// TwinCAT 3 PLC project Labor_AndreasRies
// ProgramVersion: 3.1.4023.0
// libraries:
//   Lynus Energy Basic, * (Lynus AG)
//   Lynus Persistent Data V1, * (Lynus AG)
//   Lynus Standards, * (Lynus AG)
//   Tc2_IoFunctions, * (Beckhoff Automation GmbH)
//   Tc2_ModbusSrv, * (Beckhoff Automation GmbH)
//   Tc2_Standard, * (Beckhoff Automation GmbH)
//   Tc2_System, * (Beckhoff Automation GmbH)
//   Tc2_Utilities, * (Beckhoff Automation GmbH)
//   Tc3_IotBase, * (Beckhoff Automation GmbH)
//   Tc3_JsonXml, * (Beckhoff Automation GmbH)
//   Tc3_Module, * (Beckhoff Automation GmbH)
//   EfficientIO Communicator,newest,EfficientIO
// project tree:
//   / FastTask.TcTTO, MiddleTask.TcTTO, SlowTask.TcTTO (not stored)
//   FBs/ FB_Shelly_Pro2PM.TcPOU, FB_Shelly_Pro2PM_Helper.TcPOU, FB_Shelly_Pro4PM.TcPOU, FB_Shelly_Pro4PM_Helper.TcPOU
//   POUs/ FB_CurveRead.TcPOU, FB_ECS_Keba_P30.TcPOU, prgComEffIO.TcPOU, prgCS.TcPOU, prgEM.TcPOU, prgMain.TcPOU, prgPersistent.TcPOU, prgRWEffIO.TcPOU, prgVarEffIO.TcPOU, prg_SystemTime.TcPOU
// real-time tasks:
//   TASK FastTask: cycle T#5ms, priority 6, ADS port 350
//   TASK MiddleTask: cycle T#10ms, priority 8, ADS port 351
//   TASK SlowTask: cycle T#20ms, priority 10, ADS port 352
// I/O:
//   DEVICE Gerät 1 (Beckhoff CCAT)
//   DEVICE Gerät 2 (CX-BK)
//     Box 1 (CX-BK)
// variable links:
//   Labor_AndreasRies/Labor_AndreasRies Instance <-> Device 2 (CX-BK)/Box 1 (CX-BK)
//     MiddleTask Inputs/prgEM.fbEM1.fbKL3403.byStateCH1 <-> Term 2 (KL3403)/Channel 1/Status
//     MiddleTask Inputs/prgEM.fbEM1.fbKL3403.byStateCH2 <-> Term 2 (KL3403)/Channel 2/Status
//     MiddleTask Inputs/prgEM.fbEM1.fbKL3403.byStateCH3 <-> Term 2 (KL3403)/Channel 3/Status
//     MiddleTask Inputs/prgEM.fbEM1.fbKL3403.iDataInCH1 <-> Term 2 (KL3403)/Channel 1/Daten Ein
//     MiddleTask Inputs/prgEM.fbEM1.fbKL3403.iDataInCH2 <-> Term 2 (KL3403)/Channel 2/Daten Ein
//     MiddleTask Inputs/prgEM.fbEM1.fbKL3403.iDataInCH3 <-> Term 2 (KL3403)/Channel 3/Daten Ein
//     MiddleTask Inputs/prgEM.fbKBusState.uiKBusState_OUT <-> Inputs/State
//     MiddleTask Inputs/prgMain.int_Temp_1_1 <-> Term 3 (KL3204)/Channel 1/Daten Ein
//     MiddleTask Inputs/prgMain.int_Temp_1_2 <-> Term 3 (KL3204)/Channel 2/Daten Ein
//     MiddleTask Inputs/prgMain.int_Temp_1_3 <-> Term 3 (KL3204)/Channel 3/Daten Ein
//     MiddleTask Inputs/prgMain.int_Temp_1_4 <-> Term 3 (KL3204)/Channel 4/Daten Ein
//     MiddleTask Inputs/prgMain.int_Temp_2_1 <-> Term 4 (KL3204)/Channel 1/Daten Ein
//     MiddleTask Inputs/prgMain.stInData_22/iDataIn <-> Term 4 (KL3204)/Channel 2/Daten Ein
//     MiddleTask Inputs/prgMain.stInData_24/iDataIn <-> Term 4 (KL3204)/Channel 4/Daten Ein
//     MiddleTask Inputs/prgMain.stInData_22/iState <-> Term 4 (KL3204)/Channel 2/Status
//     MiddleTask Inputs/prgMain.stInData_24/iState <-> Term 4 (KL3204)/Channel 4/Status
//     MiddleTask Inputs/prgMain.stInData_W22/iDataIn <-> Term 4 (KL3204)/Channel 3/Daten Ein
//     MiddleTask Inputs/prgMain.stInData_W22/iState <-> Term 4 (KL3204)/Channel 3/Status
//     MiddleTask Outputs/prgEM.fbEM1.fbKL3403.byCntrCH1 <-> Term 2 (KL3403)/Channel 1/Kontrolle
//     MiddleTask Outputs/prgEM.fbEM1.fbKL3403.byCntrCH2 <-> Term 2 (KL3403)/Channel 2/Kontrolle
//     MiddleTask Outputs/prgEM.fbEM1.fbKL3403.byCntrCH3 <-> Term 2 (KL3403)/Channel 3/Kontrolle
//     MiddleTask Outputs/prgMain.stOutData_22/iCtrl <-> Term 4 (KL3204)/Channel 2/Kontrolle
//     MiddleTask Outputs/prgMain.stOutData_24/iCtrl <-> Term 4 (KL3204)/Channel 4/Kontrolle
//     MiddleTask Outputs/prgMain.stOutData_22/iDataOut <-> Term 4 (KL3204)/Channel 2/Daten Aus
//     MiddleTask Outputs/prgMain.stOutData_24/iDataOut <-> Term 4 (KL3204)/Channel 4/Daten Aus
//     MiddleTask Outputs/prgMain.stOutData_W22/iCtrl <-> Term 4 (KL3204)/Channel 3/Kontrolle
//     MiddleTask Outputs/prgMain.stOutData_W22/iDataOut <-> Term 4 (KL3204)/Channel 3/Daten Aus

CONFIGURATION Labor_AndreasRies
    RESOURCE PLC ON TwinCAT3
        TASK FastTask(INTERVAL := T#5ms, PRIORITY := 6);
        TASK MiddleTask(INTERVAL := T#10ms, PRIORITY := 8);
        PROGRAM prgRWEffIO WITH FastTask : prgRWEffIO;
        PROGRAM prgVarEffIO WITH FastTask : prgVarEffIO;
        PROGRAM prg_SystemTime WITH FastTask : prg_SystemTime;
        PROGRAM prgCS WITH MiddleTask : prgCS;
        PROGRAM prgEM WITH MiddleTask : prgEM;
        PROGRAM prgPersistent WITH MiddleTask : prgPersistent;
        PROGRAM prgMain WITH MiddleTask : prgMain;
    END_RESOURCE
END_CONFIGURATION

// ---- POUs/prgRWEffIO.TcPOU
PROGRAM prgRWEffIO
VAR
	fbRW1		: FB_ReadWrite_V2;
	mFirst: BOOL;
END_VAR

fbRW1(bBusy=> , bError=> , udiErrorCodeOut=> , eErrorReadWrite_Out=> );


IF mFirst=FALSE THEN
	prgRWEffIO.fbRW1.eUploadType := 4;
	mFirst:=TRUE;	
END_IF

END_PROGRAM

// ---- POUs/prgVarEffIO.TcPOU
PROGRAM prgVarEffIO
VAR
	fbVar		: FB_VarInfo;
	int_temp_1	:INT; 					//{#lynus.ag#()}
	int_temp_2	:INT; 					//{#lynus.ag#()}
	int_temp_3	:INT; 					//{#lynus.ag#()}
	int_temp_4	:INT; 					//{#lynus.ag#()}
	int_temp_5	:INT; 					//{#lynus.ag#()}
	int_temp_6	:INT; 					//{#lynus.ag#()}
	int_temp_7	:INT; 					//{#lynus.ag#()}
	int_temp_8	:INT; 					//{#lynus.ag#()}
	int_temp_9	:INT; 					//{#lynus.ag#()}
	int_temp_10	:INT; 					//{#lynus.ag#()}
	int_temp_11	:INT; 					//{#lynus.ag#()}
	int_temp_12	:INT; 					//{#lynus.ag#()}
	int_temp_13	:INT; 					//{#lynus.ag#()}
	int_temp_14	:INT; 					//{#lynus.ag#()}
	int_temp_15	:INT; 					//{#lynus.ag#()}
	int_temp_16	:INT; 					//{#lynus.ag#()}
	int_temp_17	:INT; 					//{#lynus.ag#()}
	int_temp_18	:INT; 					//{#lynus.ag#()}
	int_temp_19	:INT; 					//{#lynus.ag#()}
	int_temp_20	:INT; 					//{#lynus.ag#()}
	int_temp_21	:INT; 					//{#lynus.ag#()}
	int_temp_22	:INT; 					//{#lynus.ag#()}
	int_temp_23	:INT; 					//{#lynus.ag#()}
	int_temp_24	:INT; 					//{#lynus.ag#()}
	int_temp_25	:INT; 					//{#lynus.ag#()}
	int_temp_26	:INT; 					//{#lynus.ag#()}
	int_temp_27	:INT; 					//{#lynus.ag#()}
	int_temp_28	:INT; 					//{#lynus.ag#()}
	int_temp_29	:INT; 					//{#lynus.ag#()}
	int_temp_30	:INT; 					//{#lynus.ag#()}
	int_temp_31	:INT; 					//{#lynus.ag#()}
	int_temp_32	:INT; 					//{#lynus.ag#()}
	int_temp_33	:INT; 					//{#lynus.ag#()}
	int_temp_34	:INT; 					//{#lynus.ag#()}
	int_temp_35	:INT; 					//{#lynus.ag#()}
	int_temp_36	:INT; 					//{#lynus.ag#()}
	int_temp_37	:INT; 					//{#lynus.ag#()}
	int_temp_38	:INT; 					//{#lynus.ag#()}
	int_temp_39	:INT; 					//{#lynus.ag#()}
	int_temp_40	:INT; 					//{#lynus.ag#()}
	int_temp_41	:INT; 					//{#lynus.ag#()}
	int_temp_42	:INT; 					//{#lynus.ag#()}
	int_temp_43	:INT; 					//{#lynus.ag#()}
	int_temp_44	:INT; 					//{#lynus.ag#()}
	int_temp_45	:INT; 					//{#lynus.ag#()}
	int_temp_46	:INT; 					//{#lynus.ag#()}
	int_temp_47	:INT; 					//{#lynus.ag#()}
	int_temp_48	:INT; 					//{#lynus.ag#()}
	int_temp_49	:INT; 					//{#lynus.ag#()}
	int_temp2_1	:INT; 					//{#lynus.ag#()}
	int_temp2_2	:INT; 					//{#lynus.ag#()}
	int_temp2_3	:INT; 					//{#lynus.ag#()}
	int_temp2_4	:INT; 					//{#lynus.ag#()}
	int_temp2_5	:INT; 					//{#lynus.ag#()}
	int_temp2_6	:INT; 					//{#lynus.ag#()}
	int_temp2_7	:INT; 					//{#lynus.ag#()}
	int_temp2_8	:INT; 					//{#lynus.ag#()}
	int_temp2_9	:INT; 					//{#lynus.ag#()}
	int_temp2_10	:INT; 					//{#lynus.ag#()}
	int_temp2_11	:INT; 					//{#lynus.ag#()}
	int_temp2_12	:INT; 					//{#lynus.ag#()}
	int_temp2_13	:INT; 					//{#lynus.ag#()}
	int_temp2_14	:INT; 					//{#lynus.ag#()}
	int_temp2_15	:INT; 					//{#lynus.ag#()}
	int_temp2_16	:INT; 					//{#lynus.ag#()}
	int_temp2_17	:INT; 					//{#lynus.ag#()}
	int_temp2_18	:INT; 					//{#lynus.ag#()}
	int_temp2_19	:INT; 					//{#lynus.ag#()}
	int_temp2_20	:INT; 					//{#lynus.ag#()}
	int_temp2_21	:INT; 					//{#lynus.ag#()}
	int_temp2_22	:INT; 					//{#lynus.ag#()}
	int_temp2_23	:INT; 					//{#lynus.ag#()}
	int_temp2_24	:INT; 					//{#lynus.ag#()}
	int_temp2_25	:INT; 					//{#lynus.ag#()}
	int_temp2_26	:INT; 					//{#lynus.ag#()}
	int_temp2_27	:INT; 					//{#lynus.ag#()}
	int_temp2_28	:INT; 					//{#lynus.ag#()}
	int_temp2_29	:INT; 					//{#lynus.ag#()}
	int_temp2_30	:INT; 					//{#lynus.ag#()}
	int_temp2_31	:INT; 					//{#lynus.ag#()}
	int_temp2_32	:INT; 					//{#lynus.ag#()}
	int_temp2_33	:INT; 					//{#lynus.ag#()}
	int_temp2_34	:INT; 					//{#lynus.ag#()}
	int_temp2_35	:INT; 					//{#lynus.ag#()}
	int_temp2_36	:INT; 					//{#lynus.ag#()}
	int_temp2_37	:INT; 					//{#lynus.ag#()}
	int_temp2_38	:INT; 					//{#lynus.ag#()}
	int_temp2_39	:INT; 					//{#lynus.ag#()}
	int_temp2_40	:INT; 					//{#lynus.ag#()}
	int_temp2_41	:INT; 					//{#lynus.ag#()}
	int_temp2_42	:INT; 					//{#lynus.ag#()}
	int_temp2_43	:INT; 					//{#lynus.ag#()}
	int_temp2_44	:INT; 					//{#lynus.ag#()}
	int_temp2_45	:INT; 					//{#lynus.ag#()}
	int_temp2_46	:INT; 					//{#lynus.ag#()}
	int_temp2_47	:INT; 					//{#lynus.ag#()}
	int_temp2_48	:INT; 					//{#lynus.ag#()}
	int_temp2_49	:INT; 					//{#lynus.ag#()}
	int_temp3_1	:INT; 					//{#lynus.ag#()}
	int_temp3_2	:INT; 					//{#lynus.ag#()}
	int_temp3_3	:INT; 					//{#lynus.ag#()}
	int_temp3_4	:INT; 					//{#lynus.ag#()}
	int_temp3_5	:INT; 					//{#lynus.ag#()}
	int_temp3_6	:INT; 					//{#lynus.ag#()}
	int_temp3_7	:INT; 					//{#lynus.ag#()}
	int_temp3_8	:INT; 					//{#lynus.ag#()}
	int_temp3_9	:INT; 					//{#lynus.ag#()}
	int_temp3_10	:INT; 					//{#lynus.ag#()}
	int_temp3_11	:INT; 					//{#lynus.ag#()}
	int_temp3_12	:INT; 					//{#lynus.ag#()}
	int_temp3_13	:INT; 					//{#lynus.ag#()}
	int_temp3_14	:INT; 					//{#lynus.ag#()}
	int_temp3_15	:INT; 					//{#lynus.ag#()}
	int_temp3_16	:INT; 					//{#lynus.ag#()}
	int_temp3_17	:INT; 					//{#lynus.ag#()}
	int_temp3_18	:INT; 					//{#lynus.ag#()}
	int_temp3_19	:INT; 					//{#lynus.ag#()}
	int_temp3_20	:INT; 					//{#lynus.ag#()}
	int_temp3_21	:INT; 					//{#lynus.ag#()}
	int_temp3_22	:INT; 					//{#lynus.ag#()}
	int_temp3_23	:INT; 					//{#lynus.ag#()}
	int_temp3_24	:INT; 					//{#lynus.ag#()}
	int_temp3_25	:INT; 					//{#lynus.ag#()}
	int_temp3_26	:INT; 					//{#lynus.ag#()}
	int_temp3_27	:INT; 					//{#lynus.ag#()}
	int_temp3_28	:INT; 					//{#lynus.ag#()}
	int_temp3_29	:INT; 					//{#lynus.ag#()}
	int_temp3_30	:INT; 					//{#lynus.ag#()}
	int_temp3_31	:INT; 					//{#lynus.ag#()}
	int_temp3_32	:INT; 					//{#lynus.ag#()}
	int_temp3_33	:INT; 					//{#lynus.ag#()}
	int_temp3_34	:INT; 					//{#lynus.ag#()}
	int_temp3_35	:INT; 					//{#lynus.ag#()}
	int_temp3_36	:INT; 					//{#lynus.ag#()}
	int_temp3_37	:INT; 					//{#lynus.ag#()}
	int_temp3_38	:INT; 					//{#lynus.ag#()}
	int_temp3_39	:INT; 					//{#lynus.ag#()}
	int_temp3_40	:INT; 					//{#lynus.ag#()}
	int_temp3_41	:INT; 					//{#lynus.ag#()}
	int_temp3_42	:INT; 					//{#lynus.ag#()}
	int_temp3_43	:INT; 					//{#lynus.ag#()}
	int_temp3_44	:INT; 					//{#lynus.ag#()}
	int_temp3_45	:INT; 					//{#lynus.ag#()}
	int_temp3_46	:INT; 					//{#lynus.ag#()}
	int_temp3_47	:INT; 					//{#lynus.ag#()}
	int_temp3_48	:INT; 					//{#lynus.ag#()}
	int_temp3_49	:INT; 					//{#lynus.ag#()}
	int_temp4_1	:INT; 					//{#lynus.ag#()}
	int_temp4_2	:INT; 					//{#lynus.ag#()}
	int_temp4_3	:INT; 					//{#lynus.ag#()}
	int_temp4_4	:INT; 					//{#lynus.ag#()}
	int_temp4_5	:INT; 					//{#lynus.ag#()}
	int_temp4_6	:INT; 					//{#lynus.ag#()}
	int_temp4_7	:INT; 					//{#lynus.ag#()}
	int_temp4_8	:INT; 					//{#lynus.ag#()}
	int_temp4_9	:INT; 					//{#lynus.ag#()}
	int_temp4_10	:INT; 					//{#lynus.ag#()}
	int_temp4_11	:INT; 					//{#lynus.ag#()}
	int_temp4_12	:INT; 					//{#lynus.ag#()}
	int_temp4_13	:INT; 					//{#lynus.ag#()}
	int_temp4_14	:INT; 					//{#lynus.ag#()}
	int_temp4_15	:INT; 					//{#lynus.ag#()}
	int_temp4_16	:INT; 					//{#lynus.ag#()}
	int_temp4_17	:INT; 					//{#lynus.ag#()}
	int_temp4_18	:INT; 					//{#lynus.ag#()}
	int_temp4_19	:INT; 					//{#lynus.ag#()}
	int_temp4_20	:INT; 					//{#lynus.ag#()}
	int_temp4_21	:INT; 					//{#lynus.ag#()}
	int_temp4_22	:INT; 					//{#lynus.ag#()}
	int_temp4_23	:INT; 					//{#lynus.ag#()}
	int_temp4_24	:INT; 					//{#lynus.ag#()}
	int_temp4_25	:INT; 					//{#lynus.ag#()}
	int_temp4_26	:INT; 					//{#lynus.ag#()}
	int_temp4_27	:INT; 					//{#lynus.ag#()}
	int_temp4_28	:INT; 					//{#lynus.ag#()}
	int_temp4_29	:INT; 					//{#lynus.ag#()}
	int_temp4_30	:INT; 					//{#lynus.ag#()}
	int_temp4_31	:INT; 					//{#lynus.ag#()}
	int_temp4_32	:INT; 					//{#lynus.ag#()}
	int_temp4_33	:INT; 					//{#lynus.ag#()}
	int_temp4_34	:INT; 					//{#lynus.ag#()}
	int_temp4_35	:INT; 					//{#lynus.ag#()}
	int_temp4_36	:INT; 					//{#lynus.ag#()}
	int_temp4_37	:INT; 					//{#lynus.ag#()}
	int_temp4_38	:INT; 					//{#lynus.ag#()}
	int_temp4_39	:INT; 					//{#lynus.ag#()}
	int_temp4_40	:INT; 					//{#lynus.ag#()}
	int_temp4_41	:INT; 					//{#lynus.ag#()}
	int_temp4_42	:INT; 					//{#lynus.ag#()}
	int_temp4_43	:INT; 					//{#lynus.ag#()}
	int_temp4_44	:INT; 					//{#lynus.ag#()}
	int_temp4_45	:INT; 					//{#lynus.ag#()}
	int_temp4_46	:INT; 					//{#lynus.ag#()}
	int_temp4_47	:INT; 					//{#lynus.ag#()}
	int_temp4_48	:INT; 					//{#lynus.ag#()}
	int_temp4_49	:INT; 					//{#lynus.ag#()}
	m_test: BOOL;
	mtest: BOOL;
END_VAR

fbVar(
	bReadInfo:= , 
	eTMCFile:= eSelectTMCFile.eDontUseTMCFile, 
	eSavePositionTMCFile:= eSavePositionOnPLC.ePostionHardDisk, 
	udiCounterFoundVariables=> , 
	bError=> , 
	bBusy=> , 
	byProgress=> , 
	udiErrorCodeOut=> , 
	eErrorVarInfo_Out=> , 
	sVarWithError=> );
IF mtest THEN
	int_temp_1 := 	int_temp_1+1;
	int_temp_2 := 	int_temp_2+10;
	int_temp_3 := 	int_temp_3+100;
	int_temp_4 := 	int_temp_4+1000;
	int_temp_5 := 	int_temp_5-1;
	int_temp_6 := 	int_temp_6-10;
	int_temp_7 := 	int_temp_7-100;
	int_temp_8 := 	int_temp_8-1000;
	int_temp_9 := 	int_temp_9+2;
	int_temp_10 := 	int_temp_10+5;
	int_temp_11 := 	int_temp_1;
	int_temp_12 := 	int_temp_2;
	int_temp_13 := 	int_temp_3;
	int_temp_14 := 	int_temp_4;
	int_temp_15 := 	int_temp_5;
	int_temp_16 := 	int_temp_6;
	int_temp_17 := 	int_temp_7;
	int_temp_18 := 	int_temp_8;
	int_temp_19 := 	int_temp_9;
	int_temp_20 := 	int_temp_10;
	int_temp_21 := 	int_temp_1;
	int_temp_22 := 	int_temp_2;
	int_temp_23 := 	int_temp_3;
	int_temp_24 := 	int_temp_4;
	int_temp_25 := 	int_temp_5;
	int_temp_26 := 	int_temp_6;
	int_temp_27 := 	int_temp_7;
	int_temp_28 := 	int_temp_8;
	int_temp_29 := 	int_temp_9;
	int_temp_30 := 	int_temp_10;
	int_temp_31 := 	int_temp_1;
	int_temp_32 := 	int_temp_2;
	int_temp_33 := 	int_temp_3;
	int_temp_34 := 	int_temp_4;
	int_temp_35 := 	int_temp_5;
	int_temp_36 := 	int_temp_6;
	int_temp_37 := 	int_temp_7;
	int_temp_38 := 	int_temp_8;
	int_temp_39 := 	int_temp_9;
	int_temp_40 := 	int_temp_10;
	int_temp_41 := 	int_temp_1;
	int_temp_42 := 	int_temp_2;
	int_temp_43 := 	int_temp_3;
	int_temp_44 := 	int_temp_4;
	int_temp_45 := 	int_temp_5;
	int_temp_46 := 	int_temp_6;
	int_temp_47 := 	int_temp_7;
	int_temp_48 := 	int_temp_8;
	int_temp_49 := 	int_temp_9;
	int_temp2_1 := 	int_temp2_1+1;
	int_temp2_2 := 	int_temp2_2+10;
	int_temp2_3 := 	int_temp2_3+100;
	int_temp2_4 := 	int_temp2_4+1000;
	int_temp2_5 := 	int_temp2_5-1;
	int_temp2_6 := 	int_temp2_6-10;
	int_temp2_7 := 	int_temp2_7-100;
	int_temp2_8 := 	int_temp2_8-1000;
	int_temp2_9 := 	int_temp2_9+2;
	int_temp2_10 := 	int_temp2_10+5;
	int_temp2_11 := 	int_temp2_1;
	int_temp2_12 := 	int_temp2_2;
	int_temp2_13 := 	int_temp2_3;
	int_temp2_14 := 	int_temp2_4;
	int_temp2_15 := 	int_temp2_5;
	int_temp2_16 := 	int_temp2_6;
	int_temp2_17 := 	int_temp2_7;
	int_temp2_18 := 	int_temp2_8;
	int_temp2_19 := 	int_temp2_9;
	int_temp2_20 := 	int_temp2_10;
	int_temp2_21 := 	int_temp2_1;
	int_temp2_22 := 	int_temp2_2;
	int_temp2_23 := 	int_temp2_3;
	int_temp2_24 := 	int_temp2_4;
	int_temp2_25 := 	int_temp2_5;
	int_temp2_26 := 	int_temp2_6;
	int_temp2_27 := 	int_temp2_7;
	int_temp2_28 := 	int_temp2_8;
	int_temp2_29 := 	int_temp2_9;
	int_temp2_30 := 	int_temp2_10;
	int_temp2_31 := 	int_temp2_1;
	int_temp2_32 := 	int_temp2_2;
	int_temp2_33 := 	int_temp2_3;
	int_temp2_34 := 	int_temp2_4;
	int_temp2_35 := 	int_temp2_5;
	int_temp2_36 := 	int_temp2_6;
	int_temp2_37 := 	int_temp2_7;
	int_temp2_38 := 	int_temp2_8;
	int_temp2_39 := 	int_temp2_9;
	int_temp2_40 := 	int_temp2_10;
	int_temp2_41 := 	int_temp2_1;
	int_temp2_42 := 	int_temp2_2;
	int_temp2_43 := 	int_temp2_3;
	int_temp2_44 := 	int_temp2_4;
	int_temp2_45 := 	int_temp2_5;
	int_temp2_46 := 	int_temp2_6;
	int_temp2_47 := 	int_temp2_7;
	int_temp2_48 := 	int_temp2_8;
	int_temp2_49 := 	int_temp2_9;
	int_temp3_1 := 	int_temp3_1+1;
	int_temp3_2 := 	int_temp3_2+10;
	int_temp3_3 := 	int_temp3_3+100;
	int_temp3_4 := 	int_temp3_4+1000;
	int_temp3_5 := 	int_temp3_5-1;
	int_temp3_6 := 	int_temp3_6-10;
	int_temp3_7 := 	int_temp3_7-100;
	int_temp3_8 := 	int_temp3_8-1000;
	int_temp3_9 := 	int_temp3_9+2;
	int_temp3_10 := 	int_temp3_10+5;
	int_temp3_11 := 	int_temp3_1;
	int_temp3_12 := 	int_temp3_2;
	int_temp3_13 := 	int_temp3_3;
	int_temp3_14 := 	int_temp3_4;
	int_temp3_15 := 	int_temp3_5;
	int_temp3_16 := 	int_temp3_6;
	int_temp3_17 := 	int_temp3_7;
	int_temp3_18 := 	int_temp3_8;
	int_temp3_19 := 	int_temp3_9;
	int_temp3_20 := 	int_temp3_10;
	int_temp3_21 := 	int_temp3_1;
	int_temp3_22 := 	int_temp3_2;
	int_temp3_23 := 	int_temp3_3;
	int_temp3_24 := 	int_temp3_4;
	int_temp3_25 := 	int_temp3_5;
	int_temp3_26 := 	int_temp3_6;
	int_temp3_27 := 	int_temp3_7;
	int_temp3_28 := 	int_temp3_8;
	int_temp3_29 := 	int_temp3_9;
	int_temp3_30 := 	int_temp3_10;
	int_temp3_31 := 	int_temp3_1;
	int_temp3_32 := 	int_temp3_2;
	int_temp3_33 := 	int_temp3_3;
	int_temp3_34 := 	int_temp3_4;
	int_temp3_35 := 	int_temp3_5;
	int_temp3_36 := 	int_temp3_6;
	int_temp3_37 := 	int_temp3_7;
	int_temp3_38 := 	int_temp3_8;
	int_temp3_39 := 	int_temp3_9;
	int_temp3_40 := 	int_temp3_10;
	int_temp3_41 := 	int_temp3_1;
	int_temp3_42 := 	int_temp3_2;
	int_temp3_43 := 	int_temp3_3;
	int_temp3_44 := 	int_temp3_4;
	int_temp3_45 := 	int_temp3_5;
	int_temp3_46 := 	int_temp3_6;
	int_temp3_47 := 	int_temp3_7;
	int_temp3_48 := 	int_temp3_8;
	int_temp3_49 := 	int_temp3_9;
	int_temp4_1 := 	int_temp4_1+1;
	int_temp4_2 := 	int_temp4_2+10;
	int_temp4_3 := 	int_temp4_3+100;
	int_temp4_4 := 	int_temp4_4+1000;
	int_temp4_5 := 	int_temp4_5-1;
	int_temp4_6 := 	int_temp4_6-10;
	int_temp4_7 := 	int_temp4_7-100;
	int_temp4_8 := 	int_temp4_8-1000;
	int_temp4_9 := 	int_temp4_9+2;
	int_temp4_10 := 	int_temp4_10+5;
	int_temp4_11 := 	int_temp4_1;
	int_temp4_12 := 	int_temp4_2;
	int_temp4_13 := 	int_temp4_3;
	int_temp4_14 := 	int_temp4_4;
	int_temp4_15 := 	int_temp4_5;
	int_temp4_16 := 	int_temp4_6;
	int_temp4_17 := 	int_temp4_7;
	int_temp4_18 := 	int_temp4_8;
	int_temp4_19 := 	int_temp4_9;
	int_temp4_20 := 	int_temp4_10;
	int_temp4_21 := 	int_temp4_1;
	int_temp4_22 := 	int_temp4_2;
	int_temp4_23 := 	int_temp4_3;
	int_temp4_24 := 	int_temp4_4;
	int_temp4_25 := 	int_temp4_5;
	int_temp4_26 := 	int_temp4_6;
	int_temp4_27 := 	int_temp4_7;
	int_temp4_28 := 	int_temp4_8;
	int_temp4_29 := 	int_temp4_9;
	int_temp4_30 := 	int_temp4_10;
	int_temp4_31 := 	int_temp4_1;
	int_temp4_32 := 	int_temp4_2;
	int_temp4_33 := 	int_temp4_3;
	int_temp4_34 := 	int_temp4_4;
	int_temp4_35 := 	int_temp4_5;
	int_temp4_36 := 	int_temp4_6;
	int_temp4_37 := 	int_temp4_7;
	int_temp4_38 := 	int_temp4_8;
	int_temp4_39 := 	int_temp4_9;
	int_temp4_40 := 	int_temp4_10;
	int_temp4_41 := 	int_temp4_1;
	int_temp4_42 := 	int_temp4_2;
	int_temp4_43 := 	int_temp4_3;
	int_temp4_44 := 	int_temp4_4;
	int_temp4_45 := 	int_temp4_5;
	int_temp4_46 := 	int_temp4_6;
	int_temp4_47 := 	int_temp4_7;
	int_temp4_48 := 	int_temp4_8;
	int_temp4_49 := 	int_temp4_9;
END_IF

END_PROGRAM

// ---- POUs/prg_SystemTime.TcPOU
PROGRAM prg_SystemTime
VAR
	fbNTGetSystemTime: NT_GetTime;
	intStateSystemTime: INT;
	structSystemTime: timestruct;
	stringSystemTime: STRING(19);
	stringSystemTime_ms: STRING(23);
	stringSystemDate: STRING(10);
	stringTimeOnly_ms: STRING(12);
	stringTimeOnly: STRING(8);
	stringMonth: STRING(4);
	strTimeStampEventrecorder: STRING;
END_VAR

(* get system time *)
CASE intStateSystemTime OF
	0:	fbNTGetSystemTime(Start:=FALSE);
		intStateSystemTime:=20;
	20:	fbNTGetSystemTime(Start:=TRUE);
		intStateSystemTime:=30;
	30:	fbNTGetSystemTime();
		IF NOT fbNTGetSystemTime.BUSY THEN
			structSystemTime:=fbNTGetSystemTime.TIMESTR;
			intStateSystemTime:=40;
		END_IF
	40:	intStateSystemTime:=0;
		stringSystemTime := SYSTEMTIME_TO_STRING(IN := structSystemTime);
		stringSystemTime_ms := SYSTEMTIME_TO_STRING(IN := structSystemTime);
		stringSystemDate := SYSTEMTIME_TO_STRING(IN := structSystemTime);
		stringTimeOnly_ms:=RIGHT(stringSystemTime_ms,12);
		stringTimeOnly:=RIGHT(stringSystemTime,8);
		CASE structSystemTime.wMonth OF
			1:	stringMonth:='Jan';
			2:	stringMonth:='Feb';
			3:	stringMonth:='Mae';
			4:	stringMonth:='Apr';
			5:	stringMonth:='Mai';
			6:	stringMonth:='Jun';
			7:	stringMonth:='Jul';
			8:	stringMonth:='Aug';
			9:	stringMonth:='Sep';
			10:	stringMonth:='Okt';
			11:	stringMonth:='Nov';
			12:	stringMonth:='Dez';
		END_CASE
		strTimeStampEventrecorder := CONCAT(WORD_TO_STRING(structSystemTime.wYear),stringMonth);
		IF structSystemTime.wDay <10 THEN
			strTimeStampEventrecorder := CONCAT(strTimeStampEventrecorder,'0');
		END_IF
		strTimeStampEventrecorder := CONCAT(strTimeStampEventrecorder,WORD_TO_STRING(structSystemTime.wDay));
		strTimeStampEventrecorder := CONCAT(strTimeStampEventrecorder,' ');
		IF structSystemTime.wHour <10 THEN
			strTimeStampEventrecorder := CONCAT(strTimeStampEventrecorder,'0');
		END_IF
		strTimeStampEventrecorder := CONCAT(strTimeStampEventrecorder,WORD_TO_STRING(structSystemTime.wHour));
		strTimeStampEventrecorder := CONCAT(strTimeStampEventrecorder,':');
		IF structSystemTime.wMinute <10 THEN
			strTimeStampEventrecorder := CONCAT(strTimeStampEventrecorder,'0');
		END_IF
		strTimeStampEventrecorder := CONCAT(strTimeStampEventrecorder,WORD_TO_STRING(structSystemTime.wMinute));
		strTimeStampEventrecorder := CONCAT(strTimeStampEventrecorder,':');
		IF structSystemTime.wSecond <10 THEN
			strTimeStampEventrecorder := CONCAT(strTimeStampEventrecorder,'0');
		END_IF
		strTimeStampEventrecorder := CONCAT(strTimeStampEventrecorder,WORD_TO_STRING(structSystemTime.wSecond));
		strTimeStampEventrecorder := CONCAT(strTimeStampEventrecorder,'.');
		IF structSystemTime.wMilliseconds <10 THEN
			strTimeStampEventrecorder := CONCAT(strTimeStampEventrecorder,'00');
		ELSIF structSystemTime.wMilliseconds <100 THEN
			strTimeStampEventrecorder := CONCAT(strTimeStampEventrecorder,'0');
		END_IF
		strTimeStampEventrecorder := CONCAT(strTimeStampEventrecorder,WORD_TO_STRING(structSystemTime.wMilliseconds));
END_CASE

END_PROGRAM

// ---- POUs/prgCS.TcPOU
PROGRAM prgCS
VAR
	fbCS1	:	FB_ECS_Keba_P30;
	bEnableCS1	: BOOL:=TRUE;
	
	lr_KEBA_TotalPower_KebaP30: LREAL;		//{#lynus.ag#()}
	b_KEBA_CarConnected: BOOL;				//{#lynus.ag#()}
	b_KEBA_Enabled: BOOL;					//{#lynus.ag#()}
	b_KEBA_OutputOn: BOOL;					//{#lynus.ag#()}
	dw_KEBA_ChargingState: DWORD;			//{#lynus.ag#()}
	dw_KEBA_ErrorCode: DWORD;				//{#lynus.ag#()}
	lreal_KEBA_TotalEnergyConsumption: LREAL;	//{#lynus.ag#()}
	lreal_KEBA_EnergySession: LREAL;		//{#lynus.ag#()}
	r_trig_Errror	:r_trig;
	iCount: INT;
	Str_IP: STRING(25):='192.168.1.195';
	i_ErrorCount: INT;
END_VAR
VAR PERSISTENT
	lreal_KEBA_Energy_Current_Month		: LREAL;	//{#lynus.ag#()}
	lreal_KEBA_Energy_Last_Month		: LREAL;	//{#lynus.ag#()}
	wMonthOld:WORD;
END_VAR

fbCS1(
	bEnable:= bEnableCS1, 
	bPowerDataInvers:=TRUE , 
	byElectricFuseLine:= ,
	uiFailsafeCurrent:=32000,
	uiFailsafeTimeOut:=600,
	diNrOfEMS_IN:= , 
	diNrOfEM_IN_CS:= , 
	sIPAdress:= Str_IP,        //'192.168.1.194', // DHCP zugewiesen am 11.04.2023
	stSetupECS:= , 
	stDataECS=> , 
	diNrOfECS_OUT=> , 
	lrTotalPowerECSRealTime=> );
	
	
	lr_KEBA_TotalPower_KebaP30 		:=	fbCS1.lrTotalPowerECSRealTime;
	b_KEBA_CarConnected			 	:=	fbCS1.stDataECS.bCarConnected;
	b_KEBA_Enabled					:= 	fbCS1.stDataECS.bEnabled;
	b_KEBA_OutputOn					:=	fbCS1.stDataECS.bOutputOnOff;
	dw_KEBA_ChargingState			:=  fbCs1.dwChargingState;
	dw_KEBA_ErrorCode				:=  fbCs1.dwErrorCode;
	lreal_KEBA_TotalEnergyConsumption	:=	fbCS1.lrTotalCounterEnergy_Consumption;
	lreal_KEBA_EnergySession		:=	fbCS1.lrChargedEnergySession;


// kWh current month / last month
IF prg_SystemTime.structSystemTime.wMonth <> wMonthOld AND prg_SystemTime.structSystemTime.wDay=1 THEN
	lreal_KEBA_Energy_Last_Month:=lreal_KEBA_Energy_Current_Month;
	wMonthOld:=prg_SystemTime.structSystemTime.wMonth;
END_IF
lreal_KEBA_Energy_Current_Month := prgEM.lrEnergyKeba-lreal_KEBA_Energy_Last_Month;






// scan Modbus IP address
(*
r_trig_Errror(CLK:=fbCS1.fbMBRead_FC3.bError);

IF r_trig_Errror.Q THEN
	i_ErrorCount := i_ErrorCount+1;
	IF i_ErrorCount>10 THEN 
		i_ErrorCount:=0;
		iCount:=iCount+1;
		IF iCount <0 OR iCount >255 THEN
			iCount := 100;
		END_IF
	ELSE
		i_ErrorCount:=i_ErrorCount+1;
	END_IF
END_IF	

Str_IP := concat('192.168.1.',INT_TO_STRING(iCount));
*)

END_PROGRAM

// ---- POUs/FB_ECS_Keba_P30.TcPOU
FUNCTION_BLOCK FB_ECS_Keba_P30
VAR_INPUT PERSISTENT
	///{#lynus.ag#()} //Enable the Fuctionblock and his logic
	bEnable: BOOL;
	///With True its possible to invert all received power data from the electric meter
	bPowerDataInvers: BOOL;
	///Electric Fuse Line on wich the ECS is connected => 1 2 3 (If 0 then this charging station is not connected to a Electric Fuse Line)
	byElectricFuseLine: BYTE;
	///Failsafe Current when the connection between PLC and Charging station is interrupted. 0mA = CS Off, 6000mA - 32000mA
	uiFailsafeCurrent: UINT;
	///Failsafe Timeout when the connection between PLC and Charging station is interrupted. 10 - 600 sec
	uiFailsafeTimeOut: UINT := 10;
	///Number of EMS what control this Device.
	diNrOfEMS_IN: DINT;
	///Number of the electric meter for incoming power data. (Power Data for this Device)
	diNrOfEM_IN_CS: DINT;
	///IP Adress from the Keba charging station
	sIPAdress: STRING(15);
	///{#lynus.ag#()} //Setup charging station
	stSetupECS: ST_Setup_ECS;
END_VAR
VAR_OUTPUT
	///{#lynus.ag#()} //Electric charging station output data
	stDataECS: ST_ECS_Output;
	///Active Number from the Electric charging Function for using on other functions
	diNrOfECS_OUT: DINT;
	///Total Electric Power in kW read out directly from the Charging station. (Real time)
	lrTotalPowerECSRealTime: LREAL; 		
END_VAR
VAR
	///Function block for electric charging station
	
	fbCS: FB_ElectricChargingStation;
	///Function block to calcualte the number of the Device
	
	fbNumberDevice: FB_NumberOfDevice;
	///Digital Input from external loock signal
	fbDIExternalLock: FB_XL1XXX_DI;
	///Modbus Read Function (FC3)
	
	fbMBRead_FC3: FB_MBReadRegs;
	///Modbus Write Function (FC6)
	
	fbMBWrite_FC6: FB_MBWriteSingleReg;
	///Convert Word to Dword
	
	fbConvertWordToDword: FB_CV_WORD_TO_DWORD;
	///Timer for Delay between Requests
	
	timDelay: TON;
	///Timer for Timeout
	
	timTimeout: TON;
	///Timer to dissable the Function after Lynus_Standards.Constants_General.tTimeDissableLynusFunctions Days without connection to the Lynus Cloud
	
	timDissableFunctions: TON;
	///Timer to try reset the connection Flag on the GVL. (When somebody delete the Connection Function and make only a onlinechange)
	
	timResetConnectionOnGVL: TON;
	///Charging Time
	
	timChTimeSocket: TON;
	///Timer to start the state machine with Daley after enabling or after the system ist restartet
	
	timDelayStart: TON;
	///Timer to Close the Socket after to much Errors
	
	timCloseSocket: TON;
	///Internal positive Edge
	
	FPError_FC_3: R_TRIG;
	///Internal positive Edge
	
	FPError_FC_6: R_TRIG;
	///Internal positive Edge
	
	FPEnable: R_TRIG;
	///Function to save persistent data
	
	arrPD: ARRAY[1..16] OF FB_PersistentData_Number;
	///Function to save persistent string data
	
	fbPDString: FB_PersistentData_String;
	///Buffer with Data from FC3
	
	arrBuffer_FC3: ARRAY[1..2] OF WORD;
	///Error State from the charging station
	
	bErrorCS: BOOL;
	///Modbus TCP Function Error Counter																	
	
	byMBTCPErrorCounter: BYTE;
	///Wait in Step before start to clean data on PLC
	
	byWaitInStep: BYTE;
	///State machine to handle the data on the GVL
	
	iStateGVLData: INT;
	///State machine for read out Data over Modbus TCP
	
	iStateModbusRead: INT;
	///State machine for write Data over Modbus TCP
	
	iStateModbusWrite: INT;
	///State machine for error out Data over Modbus TCP	
	
	iStateModbusError: INT;
	///Variable to compare the state machine variable to set or reset the timeout timer
	
	iStateModbus_CP: INT;
	///Number of active batterys
	
	diNumberOfActiveBatterys: DINT;
	///Number of battery inverters that work in Emergency Power operation 
	
	diNumberOfBatteryInverterInEPO: DINT;
	///Loop to clean old data on GVL
	
	diLPForGVL: DINT;
	///Counter to clean old data on GVL
	
	diCounterForGVL: DINT;
	///Sum of the SOC from all batterys
	
	dwSumSOC: DWORD;
	///Charging State from the Keba Charger
	
	dwChargingState: DWORD;
	///Cable State from the Keba Charger
	
	dwCableState: DWORD;
	///Error Code from the Keba Charger
	
	dwErrorCode: DWORD;
	///Power from the ECS in W 
	
	rPowerECS: REAL;
	///Energy Counter Consumption in Wh
	
	lrTotalCounterEnergy_Consumption: LREAL;
	///Charged Energy from the active Session in Wh
	
	lrChargedEnergySession: LREAL;
	///Loop to check some data from batterys
	
	liLPBatteryData: LINT;
	///Loop to check if 1 or more battery inverters build a island grid
	
	liLPInEPO: LINT;
	i: INT;
	word_MBadress: WORD;
END_VAR
VAR PERSISTENT
	///Number of EMS what control this Device to compare with the original
	{attribute 'conditionalshow' := ''}
	diNrOfEMS_IN_CP: DINT;
END_VAR

//Creator : Kai Ebensperger
//Company : Lynus AG
//Date : 15.07.2022
//Version : 1.0.0.0

//With this Funcition its possible to communicate with a Keba P30 Charging station over Modbus TCP.
//Support the C-Series from Version 3.10.16 or higher
//Support the X-Series from Version 1.11 or higher
//Its possible to controll the charging station over the charge current
//When the Function send 0 Ampere is switched of, then the charging station is blocked and its not possible to charge
//The Communication is not so fast because in the Documentation they write that we can read every 500MS but we can write onle ever 5 seconds.
//We can read only 1 Register at each command. Its not possible to read more Registers with 1 command
//The Unit ID is always 255
//Also the Settings for Fail Save is includes in ths Fuction. The Failsave Current is set to uiFailsafeCurrent.
//Failsafe takes effect when the connection between the PLC and the charging station is interrupted. Timout is uiFailsafeTimeOut in seconds.

//Versions that are supported : 1.3

//NOTE for diNr.....Designation => 
//_IN = Here Data come in from other Functions or go out to other functions about the GVL
//_OUT = Here Data go out to other functions about the GVL

(*--------------------------------------------------------------------------------------------Limits-------------------------------------------------------------------------------------*)

diNrOfEMS_IN := LIMIT(0,diNrOfEMS_IN,Constants_Energy.diMaxNumberOfEMS);
	diNrOfEM_IN_CS := LIMIT(0,diNrOfEM_IN_CS,Constants_Energy.diMaxNumberOfElectricMeters);
		byElectricFuseLine := LIMIT(0,byElectricFuseLine,30);
			IF uiFailsafeCurrent > 0 THEN 
				uiFailsafeCurrent := LIMIT(6000,uiFailsafeCurrent,32000);
			END_IF 
				uiFailsafeTimeOut := LIMIT(10,uiFailsafeTimeOut,600);	
		
(*------------------------------------------------------------------Power Data----------------------------------------------------------------------------*)

IF diNrOfEM_IN_CS <> 0 THEN
	//Energy Session Input data
	fbCS.bCalculateEnergySession := FALSE;
	fbCS.arrSocketPowerECS[1] := 0;
	fbCS.arrSocketPowerECS[2] := 0;
	fbCS.arrSocketPowerECS[3] := 0;
	fbCS.arrSocketPowerECS[4] := 0;
	fbCS.arrSocketEnergySession[1] := 0;
	fbCS.arrSocketEnergySession[2] := 0;
	fbCS.arrSocketEnergySession[3] := 0;
	fbCS.arrSocketEnergySession[4] := 0;
		IF NOT bPowerDataInvers THEN
			//Energy meter input data for cs Function block
			fbCS.lrCounterEnergyT1_Consumption := Lynus_Standards.GVL_Energy.stDataElectricMeters[diNrOfEM_IN_CS].lrCounterEnergyT1_Production * 1000;
			fbCS.lrCounterEnergyT2_Consumption := Lynus_Standards.GVL_Energy.stDataElectricMeters[diNrOfEM_IN_CS].lrCounterEnergyT2_Production * 1000;
			fbCS.lrCounterEnergyT1_Production := Lynus_Standards.GVL_Energy.stDataElectricMeters[diNrOfEM_IN_CS].lrCounterEnergyT1_Consumption * 1000;
			fbCS.lrCounterEnergyT2_Production := Lynus_Standards.GVL_Energy.stDataElectricMeters[diNrOfEM_IN_CS].lrCounterEnergyT1_Consumption * 1000;
			fbCS.lrTotalCounterEnergy_Consumption := Lynus_Standards.GVL_Energy.stDataElectricMeters[diNrOfEM_IN_CS].lrTotalCounterEnergy_Production * 1000;
			fbCS.lrTotalCounterEnergy_Production := Lynus_Standards.GVL_Energy.stDataElectricMeters[diNrOfEM_IN_CS].lrTotalCounterEnergy_Consumption * 1000;
				fbCS.lrTotalPowerECS := (Lynus_Standards.GVL_Energy.stDataElectricMeters[diNrOfEM_IN_CS].lrPower * 1000) * -1;
			ELSE
			//Energy meter input data for cs Function block
			fbCS.lrCounterEnergyT1_Consumption := Lynus_Standards.GVL_Energy.stDataElectricMeters[diNrOfEM_IN_CS].lrCounterEnergyT1_Consumption * 1000;
			fbCS.lrCounterEnergyT2_Consumption := Lynus_Standards.GVL_Energy.stDataElectricMeters[diNrOfEM_IN_CS].lrCounterEnergyT2_Consumption * 1000;
			fbCS.lrCounterEnergyT1_Production := Lynus_Standards.GVL_Energy.stDataElectricMeters[diNrOfEM_IN_CS].lrCounterEnergyT1_Production * 1000;
			fbCS.lrCounterEnergyT2_Production := Lynus_Standards.GVL_Energy.stDataElectricMeters[diNrOfEM_IN_CS].lrCounterEnergyT2_Production * 1000;
			fbCS.lrTotalCounterEnergy_Consumption := Lynus_Standards.GVL_Energy.stDataElectricMeters[diNrOfEM_IN_CS].lrTotalCounterEnergy_Consumption * 1000;
			fbCS.lrTotalCounterEnergy_Production := Lynus_Standards.GVL_Energy.stDataElectricMeters[diNrOfEM_IN_CS].lrTotalCounterEnergy_Production * 1000;
				fbCS.lrTotalPowerECS := Lynus_Standards.GVL_Energy.stDataElectricMeters[diNrOfEM_IN_CS].lrPower * 1000;
		END_IF
ELSE
	//Energy meter input data for cs Function block
	fbCS.lrCounterEnergyT1_Consumption := lrTotalCounterEnergy_Consumption;
	fbCS.lrCounterEnergyT2_Consumption := 0;
	fbCS.lrCounterEnergyT1_Production := 0;
	fbCS.lrCounterEnergyT2_Production := 0;
	fbCS.lrTotalCounterEnergy_Consumption := lrTotalCounterEnergy_Consumption;
	fbCS.lrTotalCounterEnergy_Production := 0;
		fbCS.lrTotalPowerECS := rPowerECS;
	//Energy Session Input data
	fbCS.bCalculateEnergySession := FALSE;
	fbCS.arrSocketPowerECS[1] := rPowerECS;
	fbCS.arrSocketPowerECS[2] := 0;
	fbCS.arrSocketPowerECS[3] := 0;
	fbCS.arrSocketPowerECS[4] := 0;
	fbCS.arrSocketEnergySession[1] := lrChargedEnergySession;
	fbCS.arrSocketEnergySession[2] := 0;
	fbCS.arrSocketEnergySession[3] := 0;
	fbCS.arrSocketEnergySession[4] := 0;
END_IF			

(*-------------------------------------------------------------Calcualte the number of ECS---------------------------------------------------------------*)

fbNumberDevice(
	diActualNumberOfDevices:= Lynus_Standards.GVL_Energy.stNumberOfDevices.diNumberOfECS, 
	diMaxNumberOfDevices:= Constants_Energy.diMaxNumberOfElectricChargingStations, 
	udiCounterOnlineChange:= TwinCAT_SystemInfoVarList._AppInfo.OnlineChangeCnt, 
	bNumberIsCalculatet=> , 
	bFPNumberIsCalculatet=> , 
	bOnlineChange=> , 
	diNumberForThisDevice=> diNrOfECS_OUT, 
	diNumberOfTotalDevices=> );

//Write new Numer on GVL
IF fbNumberDevice.bFPNumberIsCalculatet THEN
	Lynus_Standards.GVL_Energy.stNumberOfDevices.diNumberOfECS := fbNumberDevice.diNumberOfTotalDevices;	
END_IF 

//Delete old Number on GVL
IF fbNumberDevice.bOnlineChange THEN 
	Lynus_Standards.GVL_Energy.stNumberOfDevices.diNumberOfECS := diNrOfECS_OUT;	
		iStateGVLData := 1;
END_IF

(*-------------------------------------------------------------Service from Backend is ready and check the connection to backen for dissabel/enable Function---------------------------------------------------------------*)

//Try to reset the variable for connection on the GVL. When all is normal then the Lynus Mqtt connection function set this variable to true in the next cycle
//When we have no connection to the backend then after Lynus_Standards.Constants_General.tTimeDissableLynusFunctions days the Function is dissabled with all of his functionalities
timResetConnectionOnGVL(IN:= NOT timResetConnectionOnGVL.Q, PT:= T#1H, Q=> , ET=> );
	IF timResetConnectionOnGVL.Q THEN Lynus_Standards.GVL_Communicator.bStateConnectionToEnableFunctions := FALSE; END_IF
		IF NOT Lynus_Standards.GVL_Communicator.bStateConnectionToEnableFunctions THEN timDissableFunctions.IN := TRUE; ELSE timDissableFunctions.IN := FALSE; END_IF  
			timDissableFunctions(IN:= , PT:= Lynus_Standards.Constants_General.tTimeDissableLynusFunctions, Q=> , ET=> );
			
(*--------------------------------------------------------------------------------------------State Machine Read--------------------------------------------------------------------------------------*)

//Timer for Delay
timDelay(IN:= , PT:= T#750MS, Q=> , ET=> );

//Timer for Timeout in Statemachine
IF (iStateModbusRead > 0 AND iStateModbusRead <= 7 AND iStateModbusRead = iStateModbus_CP) OR
		(iStateModbusWrite > 0 AND iStateModbusWrite <= 2 AND iStateModbusWrite = iStateModbus_CP) THEN
			timTimeout.IN := TRUE;
ELSE	
			timTimeout.IN := FALSE;
END_IF
	//Timeout Timer is dissabled when the Init Step is aktiv or the function is not enabled
	IF (iStateModbusRead = 0 AND iStateModbusWrite = 0) OR NOT bEnable THEN timTimeout.IN := FALSE; END_IF
		timTimeout(IN:= , PT:= T#10S, Q=> , ET=> );

//Enable with Delay that not all sockets have to be created at the same time
timDelayStart(IN:= bEnable, PT:= T#20MS * diNrOfECS_OUT, Q=> , ET=> );
	FPEnable(CLK:= timDelayStart.Q, Q=> );

IF FPEnable.Q AND iStateModbusRead = 0 AND iStateModbusWrite = 0 THEN iStateModbusRead := 1; END_IF		
		
//Not Enabled
IF NOT bEnable THEN iStateModbusRead := 0; iStateModbusError := 0; iStateModbusWrite := 0; END_IF		
		
CASE iStateModbusRead OF
	 
	0://Init Step 
		iStateModbus_CP := 0;
			timDelay.IN := FALSE;
				fbMBRead_FC3.bExecute := FALSE;
					fbMBWrite_FC6.bExecute := FALSE;
						rPowerECS := 0;
							dwChargingState := 0;
								dwCableState := 0;	
									lrChargedEnergySession := 0;
	
	1://Charging State (Register 1000) !!!!Maybe 0 or 1....test it. Then change also the other Register Adresses!!!!!
		iStateModbus_CP := iStateModbusRead;

		//Start Read
		fbMBRead_FC3.nQuantity := 2;
			fbMBRead_FC3.nMBAddr := 1000;
				fbMBRead_FC3.bExecute := TRUE;
					fbMBRead_FC3.nUnitID := 255;
			
		IF fbMBRead_FC3.bBusy THEN timDelay.IN := TRUE; END_IF
		
		//Wait for Delay, copy Data and then next step
		IF NOT fbMBRead_FC3.bBusy AND NOT fbMBRead_FC3.bError AND timDelay.Q THEN
			//Charging State
			fbConvertWordToDword(wInputValue_1:= arrBuffer_FC3[1], wInputValue_2:= arrBuffer_FC3[2], eByteOrderForConvert:= eByteOrder.eBigEndian, dwOutputValue =>);
				dwChargingState := fbConvertWordToDword.dwOutputValue;
			
			//Go to Next Step
			fbMBRead_FC3.bExecute := FALSE;
				timDelay.IN := FALSE;		
					iStateModbusRead := 2;
		END_IF	

		//Error or Timeout
		IF FPError_FC_3.Q OR timTimeout.Q THEN
			iStateModbusError := 300;
		END_IF	
		
	2://Cable State (Register 1004)
		iStateModbus_CP := iStateModbusRead;

		//Start Read
		fbMBRead_FC3.nQuantity := 2;
			fbMBRead_FC3.nMBAddr := 1004;
				fbMBRead_FC3.bExecute := TRUE;
					fbMBRead_FC3.nUnitID := 255;
			
		IF fbMBRead_FC3.bBusy THEN timDelay.IN := TRUE; END_IF
		
		//Wait for Delay, copy Data and then next step
		IF NOT fbMBRead_FC3.bBusy AND NOT fbMBRead_FC3.bError AND timDelay.Q THEN
			//Cable State
			fbConvertWordToDword(wInputValue_1:= arrBuffer_FC3[1], wInputValue_2:= arrBuffer_FC3[2], eByteOrderForConvert:= eByteOrder.eBigEndian, dwOutputValue =>);
				dwCableState := fbConvertWordToDword.dwOutputValue;
			//Go to Next Step
			fbMBRead_FC3.bExecute := FALSE;
				timDelay.IN := FALSE;		
					iStateModbusRead := 3;
		END_IF	

		//Error or Timeout
		IF FPError_FC_3.Q OR timTimeout.Q THEN
			iStateModbusError := 300;
		END_IF	
		
	3://Error Code (Register 1006)
		iStateModbus_CP := iStateModbusRead;

		//Start Read
		fbMBRead_FC3.nQuantity := 2;
			fbMBRead_FC3.nMBAddr := 1006;
				fbMBRead_FC3.bExecute := TRUE;
					fbMBRead_FC3.nUnitID := 255;
			
		IF fbMBRead_FC3.bBusy THEN timDelay.IN := TRUE; END_IF
		
		//Wait for Delay, copy Data and then next step
		IF NOT fbMBRead_FC3.bBusy AND NOT fbMBRead_FC3.bError AND timDelay.Q THEN
			//Error Code
			fbConvertWordToDword(wInputValue_1:= arrBuffer_FC3[1], wInputValue_2:= arrBuffer_FC3[2], eByteOrderForConvert:= eByteOrder.eBigEndian, dwOutputValue =>);
				dwErrorCode := fbConvertWordToDword.dwOutputValue;
			//Go to Next Step
			fbMBRead_FC3.bExecute := FALSE;
				timDelay.IN := FALSE;		
					iStateModbusRead := 4;
		END_IF	

		//Error or Timeout
		IF FPError_FC_3.Q OR timTimeout.Q THEN
			iStateModbusError := 300;
		END_IF	
		
	4://Active Power (Register 1020)
		iStateModbus_CP := iStateModbusRead;

		//Start Read
		fbMBRead_FC3.nQuantity := 2;
			fbMBRead_FC3.nMBAddr := 1020;
				fbMBRead_FC3.bExecute := TRUE;
					fbMBRead_FC3.nUnitID := 255;
			
		IF fbMBRead_FC3.bBusy THEN timDelay.IN := TRUE; END_IF
		
		//Wait for Delay, copy Data and then next step
		IF NOT fbMBRead_FC3.bBusy AND NOT fbMBRead_FC3.bError AND timDelay.Q THEN
			//Active Power in mW
			fbConvertWordToDword(wInputValue_1:= arrBuffer_FC3[1], wInputValue_2:= arrBuffer_FC3[2], eByteOrderForConvert:= eByteOrder.eBigEndian, dwOutputValue =>);
				rPowerECS := DWORD_TO_REAL(fbConvertWordToDword.dwOutputValue);
					rPowerECS := rPowerECS / 1000;	
			//Go to Next Step
			fbMBRead_FC3.bExecute := FALSE;
				timDelay.IN := FALSE;		
					iStateModbusRead := 5;
		END_IF	

		//Error or Timeout
		IF FPError_FC_3.Q OR timTimeout.Q THEN
			iStateModbusError := 300;
		END_IF	
	
	5://Total Energy (Register 1036)
		iStateModbus_CP := iStateModbusRead;

		//Start Read
		fbMBRead_FC3.nQuantity := 2;
			fbMBRead_FC3.nMBAddr := 1036;
				fbMBRead_FC3.bExecute := TRUE;
					fbMBRead_FC3.nUnitID := 255;
			
		IF fbMBRead_FC3.bBusy THEN timDelay.IN := TRUE; END_IF
		
		//Wait for Delay, copy Data and then next step
		IF NOT fbMBRead_FC3.bBusy AND NOT fbMBRead_FC3.bError AND timDelay.Q THEN
			//Total Energy in Wh
			fbConvertWordToDword(wInputValue_1:= arrBuffer_FC3[1], wInputValue_2:= arrBuffer_FC3[2], eByteOrderForConvert:= eByteOrder.eBigEndian, dwOutputValue =>);
				lrTotalCounterEnergy_Consumption := DWORD_TO_LREAL(fbConvertWordToDword.dwOutputValue);
			//Go to Next Step
			fbMBRead_FC3.bExecute := FALSE;
				timDelay.IN := FALSE;		
					iStateModbusRead := 6;
		END_IF	

		//Error or Timeout
		IF FPError_FC_3.Q OR timTimeout.Q THEN
			iStateModbusError := 300;
		END_IF	
		
	6://Charged Energy from current charging session (Register 1502)
		iStateModbus_CP := iStateModbusRead;

		//Start Read
		fbMBRead_FC3.nQuantity := 2;
			fbMBRead_FC3.nMBAddr := word_MBadress;   //1502;
				fbMBRead_FC3.bExecute := TRUE;
					fbMBRead_FC3.nUnitID := 255;
			
		IF fbMBRead_FC3.bBusy THEN timDelay.IN := TRUE; END_IF
		
		//Wait for Delay, copy Data and then next step
		IF NOT fbMBRead_FC3.bBusy AND NOT fbMBRead_FC3.bError AND timDelay.Q THEN
			//Total Energy in Wh
			fbConvertWordToDword(wInputValue_1:= arrBuffer_FC3[1], wInputValue_2:= arrBuffer_FC3[2], eByteOrderForConvert:= eByteOrder.eBigEndian, dwOutputValue =>);
				lrChargedEnergySession := DWORD_TO_LREAL(fbConvertWordToDword.dwOutputValue);
			//Go to Next Step
			fbMBRead_FC3.bExecute := FALSE;
				timDelay.IN := FALSE;		
					iStateModbusRead := 7;
		END_IF	

		//Error or Timeout
		IF FPError_FC_3.Q OR timTimeout.Q THEN
			iStateModbusError := 300;
		END_IF	
		
	7://Wait 1 Step to reset the delay counter befor start to write
		iStateModbus_CP := iStateModbusRead;
		
			// iStateModbusWrite := 1;
				//-1 because 0 is the Init Step for Read
			//	iStateModbusRead := -1;   
				iStateModbusRead := 1;   
				
			//Error on Master, changes on Inputs or Timeout
		 	IF timTimeout.Q THEN 
				iStateModbusError := 300;	 
			END_IF
	
END_CASE

(*------------------------------------------------------------------Error and Warning----------------------------------------------------------------------------*)	
 
IF dwChargingState = 4 OR dwErrorCode <> 0 THEN bErrorCS := TRUE; ELSE bErrorCS := FALSE; END_IF

IF timDissableFunctions.Q THEN fbCS.bWarning := TRUE; fbCS.iWarningCode := 0; ELSE fbCS.bWarning := FALSE; END_IF   
	IF Lynus_Standards.GVL_Energy.stNumberOfDevices.diNumberOfECS > Constants_Energy.diMaxNumberOfElectricChargingStations OR bErrorCS OR byMBTCPErrorCounter > 10 THEN 
		fbCS.bError := TRUE;
	ELSE 
		fbCS.bError := FALSE;
			fbCS.iErrorCode := 0;
	END_IF

IF Lynus_Standards.GVL_Energy.stNumberOfDevices.diNumberOfECS > Constants_Energy.diMaxNumberOfElectricChargingStations THEN fbCS.iErrorCode := 1;
ELSIF bErrorCS OR byMBTCPErrorCounter > 10 THEN fbCS.iErrorCode := 0; END_IF

(*------------------------------------------------------------------Logic----------------------------------------------------------------------------*)

//Calcualte the total SOC if we have more then 1 battery in our system
diNumberOfActiveBatterys := 0;
	dwSumSOC := 0;
		FOR liLPBatteryData := 1 TO Constants_Energy.diMaxNumberOfBatterys BY 1 DO
			IF Lynus_Standards.GVL_Energy.stDataOfBatterys[diNrOfEMS_IN,liLPBatteryData].bEnabled THEN diNumberOfActiveBatterys := diNumberOfActiveBatterys + 1; END_IF
				dwSumSOC := dwSumSOC + Lynus_Standards.GVL_Energy.stDataOfBatterys[diNrOfEMS_IN,liLPBatteryData].dwSOC;
		END_FOR
	
IF diNumberOfActiveBatterys > 0 THEN
	fbCS.dwBatterySOC := DINT_TO_DWORD(DWORD_TO_DINT(dwSumSOC) / diNumberOfActiveBatterys);
ELSE
	fbCS.dwBatterySOC := 100;	//When we have no battery in the ems system
END_IF

//Check if one or more Batterysystems or batteryinverter make island mode
diNumberOfBatteryInverterInEPO := 0;
	FOR liLPInEPO := 1 TO Constants_Energy.diMaxNumberOfBatteryInverters BY 1 DO
		IF Lynus_Standards.GVL_Energy.stDataOfBatteryInverters[diNrOfEMS_IN,liLPInEPO].bWorkOnIslandMode THEN fbCS.bEPOIsActive := TRUE; diNumberOfBatteryInverterInEPO := diNumberOfBatteryInverterInEPO + 1; END_IF
	END_FOR 
		IF diNumberOfBatteryInverterInEPO <= 0 THEN fbCS.bEPOIsActive := FALSE; END_IF

//Digital input for external lock signal
fbDIExternalLock(bInvers:= FALSE, bSignal=> );

//Car connected to the ECS
IF dwCableState = 5 OR dwCableState = 7 THEN fbCS.bCarConnected := TRUE; ELSE fbCS.bCarConnected := FALSE; END_IF

//Charging time
IF dwChargingState = 3 OR dwCableState = 7 THEN timChTimeSocket.IN := TRUE; ELSE timChTimeSocket.IN := FALSE; END_IF

IF timChTimeSocket.IN THEN fbCS.arrSocketChargingTimeInput[1] := TIME_TO_REAL(timChTimeSocket.ET) / 60000; END_IF
fbCS.arrSocketChargingTimeInput[2] := 0;
fbCS.arrSocketChargingTimeInput[3] := 0;
fbCS.arrSocketChargingTimeInput[4] := 0;

timChTimeSocket(IN:= , PT:= T#24H, Q=> , ET=> );

//Mode 3 State
//Default set to No Informantion
fbCS.arrSocketMode3StateECS[1] := '';
	//Ready or Free
	IF dwChargingState = 2 THEN fbCS.arrSocketMode3StateECS[1] := 'A'; END_IF
	//Car Connected
	IF dwCableState = 5 OR dwCableState = 7 THEN fbCS.arrSocketMode3StateECS[1] := 'B1'; END_IF
	//Charging
	IF dwChargingState = 3 OR dwCableState = 7 THEN fbCS.arrSocketMode3StateECS[1] := 'C2'; END_IF
	//Error
	IF dwChargingState = 4 OR dwErrorCode <> 0 THEN fbCS.arrSocketMode3StateECS[1] := 'F'; END_IF 

fbCS.arrSocketMode3StateECS[2] := '';
fbCS.arrSocketMode3StateECS[3] := '';
fbCS.arrSocketMode3StateECS[4] := '';

//SOC Car
fbCS.arrSOCCar[1] := 0;
fbCS.arrSOCCar[2] := 0;
fbCS.arrSOCCar[3] := 0;
fbCS.arrSOCCar[4] := 0;

//Functionblock ECS
fbCS(
	bEnable:= bEnable AND NOT timDissableFunctions.Q, 
	bError:= ,
	bWarning := ,
	bEPOIsActive:= , 
	bExternalLock:= fbDIExternalLock.bSignal, 
	bCarConnected:= , 
	bWriteWithDelay:= TRUE, 
	bCalculateEnergySession:= ,
	iErrorCode:= , 
	iWarningCode:= , 
	arrSocketChargingTimeInput:= ,
	arrSOCCar:= , 
	dwBatterySOC:= , 
	lrTotalCounterEnergy_Consumption:= , 
	lrTotalCounterEnergy_Production:= , 
	lrCounterEnergyT1_Consumption:= , 
	lrCounterEnergyT2_Consumption:= , 
	lrCounterEnergyT1_Production:= , 
	lrCounterEnergyT2_Production:= , 
	lrTotalPowerECS:= , 
	arrSocketEnergySession:= ,
	rTargetPower:= Lynus_Standards.GVL_Energy.stDataElectricChargingStations[diNrOfEMS_IN,diNrOfECS_OUT].rTargetPowerEMS, 
	rSupplyVoltage:= 692, 
	rMinCurrent:= 6, 
	tTimDelayOutput:= T#5S, 
	tDelayError:= T#5S,
	arrSocketMode3StateECS:= ,
	arrSocketPowerECS:= ,
	stSetupECS:= stSetupECS, 
	stDataECSOut=> , 
	stDataECSOutDelay=> stDataECS);

//Real time Power for Output
lrTotalPowerECSRealTime := fbCS.stDataECSOut.lrTotalPower;
	
(*------------------------------------------------------------------------------------------State Machine Write---------------------------------------------------------------------------------------------*)	

CASE iStateModbusWrite OF	

	1://Set the charging current (Reg 5004)
		iStateModbus_CP := iStateModbusWrite;
		
			fbMBWrite_FC6.nMBAddr := 5004;
				fbMBWrite_FC6.bExecute := TRUE;
					fbMBWrite_FC6.nUnitID := 255;
						//Charge Current in mA
						fbMBWrite_FC6.nValue := REAL_TO_WORD(fbCS.stDataECSOut.rTargetChargeCurrent * 1000);
		
		IF fbMBWrite_FC6.bBusy THEN timDelay.IN := TRUE; END_IF

		//Wait for Delay and then next step
		IF NOT fbMBWrite_FC6.bBusy AND NOT fbMBWrite_FC6.bError AND timDelay.Q THEN
			fbMBWrite_FC6.bExecute := FALSE;
				timDelay.IN := FALSE;
					//Go to Next Step
					iStateModbusWrite := 2;
		END_IF
				
		//Error or Timout
		IF FPError_FC_6.Q OR timTimeout.Q THEN
			iStateModbusError := 300;
		END_IF
	
	2://Enable/Dissable Charging station (Reg 5014)
		iStateModbus_CP := iStateModbusWrite;
		
			fbMBWrite_FC6.nMBAddr := 5014;
				fbMBWrite_FC6.bExecute := TRUE;
					fbMBWrite_FC6.nUnitID := 255;
						//Enable and Dissable the Charging station
						IF fbCS.stDataECSOut.rTargetChargeCurrent <> 0 THEN 
							//Enable
							fbMBWrite_FC6.nValue := 1;
						ELSE
							//Dissable
							fbMBWrite_FC6.nValue := 0;
						END_IF
		
		IF fbMBWrite_FC6.bBusy THEN timDelay.IN := TRUE; END_IF

		//Wait for Delay and then next step
		IF NOT fbMBWrite_FC6.bBusy AND NOT fbMBWrite_FC6.bError AND timDelay.Q THEN
			fbMBWrite_FC6.bExecute := FALSE;
				timDelay.IN := FALSE;
					//Go to Next Step
					iStateModbusWrite := 4; // was 3/ just for testing
		END_IF
				
		//Error or Timout
		IF FPError_FC_6.Q OR timTimeout.Q THEN
			iStateModbusError := 300;
		END_IF
		
	3://Failsafe current (Reg 5016)
		iStateModbus_CP := iStateModbusWrite;
		
			fbMBWrite_FC6.nMBAddr := 5016;
				fbMBWrite_FC6.bExecute := TRUE;
					fbMBWrite_FC6.nUnitID := 255;
						//Failsafe current in mA
						fbMBWrite_FC6.nValue := uiFailsafeCurrent;
	
		IF fbMBWrite_FC6.bBusy THEN timDelay.IN := TRUE; END_IF

		//Wait for Delay and then next step
		IF NOT fbMBWrite_FC6.bBusy AND NOT fbMBWrite_FC6.bError AND timDelay.Q THEN
			fbMBWrite_FC6.bExecute := FALSE;
				timDelay.IN := FALSE;
					//Go to Next Step
					iStateModbusWrite := 4;
		END_IF
				
		//Error or Timout
		IF FPError_FC_6.Q OR timTimeout.Q THEN
			iStateModbusError := 300;
		END_IF	
		
	4://Failsafe Timeout (Reg 5018)
		iStateModbus_CP := iStateModbusWrite;
		
			fbMBWrite_FC6.nMBAddr := 5018;
				fbMBWrite_FC6.bExecute := TRUE;
					fbMBWrite_FC6.nUnitID := 255;
						//Failsafe Timeout in sec.
						fbMBWrite_FC6.nValue := uiFailsafeTimeOut;
	
		IF fbMBWrite_FC6.bBusy THEN timDelay.IN := TRUE; END_IF

		//Wait for Delay and then next step
		IF NOT fbMBWrite_FC6.bBusy AND NOT fbMBWrite_FC6.bError AND timDelay.Q THEN
			fbMBWrite_FC6.bExecute := FALSE;
				timDelay.IN := FALSE;
					byMBTCPErrorCounter := 0; 
						//Restart from new with the Read out part
						iStateModbusRead := 1;
							iStateModbusWrite := 0;
		END_IF
				
		//Error or Timout
		IF FPError_FC_6.Q OR timTimeout.Q THEN
			iStateModbusError := 300;
		END_IF	
		
END_CASE	
	
(*------------------------------------------------------------------------------------------State Machine Error---------------------------------------------------------------------------------------------*)	

CASE iStateModbusError OF
	
	300://Error
		iStateModbus_CP := iStateModbusError;
			timDelay.IN := FALSE;
				fbMBRead_FC3.bExecute := FALSE;
					fbMBWrite_FC6.bExecute := FALSE;
						byMBTCPErrorCounter := byMBTCPErrorCounter + 1;
							byMBTCPErrorCounter := LIMIT(0,byMBTCPErrorCounter,11); 		
								//Restart from new with the Read out part after an Error
								IF byMBTCPErrorCounter < 10 THEN
									iStateModbusRead := 1;	
										iStateModbusError := 0;
											iStateModbusWrite := 0;
								ELSE
									//Wait here in the Error State for the Delay Timer and then we dont have a Timeout Error
									iStateModbusRead := -1;   // was -1
										iStateModbusWrite := - 1;
											//Start from New when the Delay is paste
											IF timCloseSocket.Q THEN
												iStateModbusRead := 1;	
													iStateModbusError := 0;
														iStateModbusWrite := 0;	
															byMBTCPErrorCounter := 0;
											END_IF
								END_IF
						
END_CASE

//Timer to close the Socket after to much TCP Errors and reopen a new one
timCloseSocket(IN:= byMBTCPErrorCounter > 10 AND fbCS.stDataECSOut.bEnabled, PT:= T#1S, Q=> , ET=> );
// was t#1m
(*------------------------------------------------------------------------------------------Modbus TCP Functions---------------------------------------------------------------------------------------------*)

fbMBRead_FC3(sIPAddr:= sIPAdress, nTCPPort:= 502,cbLength:= SIZEOF(arrBuffer_FC3), pDestAddr:= ADR(arrBuffer_FC3), tTimeout:= T#5S );
	FPError_FC_3(CLK:= fbMBRead_FC3.bError, Q=> );		

fbMBWrite_FC6(sIPAddr:= sIPAdress, nTCPPort:= 502, tTimeout:= T#5S);	
	FPError_FC_6(CLK:= fbMBWrite_FC6.bError, Q=> );

(*-----------------------------------------------------------Handle data to Global structure for electric charging stations-----------------------------------------------------------------*)

//Delte al old Data on GVL after a online change or change on the variable diNrOfEMS_IDOD
IF diNrOfEMS_IN <> diNrOfEMS_IN_CP AND iStateGVLData = 0 THEN iStateGVLData := 10; END_IF 

CASE iStateGVLData OF
	
	0://Init Step
		byWaitInStep := 0;
			diCounterForGVL := 1;
	
	1://Wait for 4 Steps before clean al Data on GVL
		byWaitInStep := byWaitInStep + 1;
			IF byWaitInStep >= 4 AND fbNumberDevice.bNumberIsCalculatet THEN iStateGVLData := 2; END_IF
				//To much Devices, back to the Init step
				IF byWaitInStep >= 4 AND NOT fbNumberDevice.bNumberIsCalculatet THEN iStateGVLData := 0; END_IF	
			
	2://Clear all Data in GVL
		FOR diLPForGVL := 1 TO Constants_Energy.diMaxNumberOfEMS BY 1 DO 
			Lynus_Standards.GVL_Energy.stDataElectricChargingStations[diLPForGVL,diCounterForGVL].bEnabled := FALSE;
				Lynus_Standards.GVL_Energy.stDataElectricChargingStations[diLPForGVL,diCounterForGVL].bIsControllable := FALSE;
					Lynus_Standards.GVL_Energy.stDataElectricChargingStations[diLPForGVL,diCounterForGVL].byErrorWarning := 0;
						Lynus_Standards.GVL_Energy.stDataElectricChargingStations[diLPForGVL,diCounterForGVL].byPriority := 0;
							Lynus_Standards.GVL_Energy.stDataElectricChargingStations[diLPForGVL,diCounterForGVL].lrPower := 0;
								Lynus_Standards.GVL_Energy.stDataElectricChargingStations[diLPForGVL,diCounterForGVL].lrPowerConsumption := 0;
									Lynus_Standards.GVL_Energy.stDataElectricChargingStations[diLPForGVL,diCounterForGVL].lrPowerProduction := 0;
										Lynus_Standards.GVL_Energy.stDataElectricChargingStations[diLPForGVL,diCounterForGVL].rMaxPower := 0;
											Lynus_Standards.GVL_Energy.stDataElectricChargingStations[diLPForGVL,diCounterForGVL].byElectricFuseLine := 0;
												//Set also the target value from ems back here to 0 and not in EMS function because EMS is in Standy when we have a online change (Problem when we delete a ems function and make a online change)
												Lynus_Standards.GVL_Energy.stDataElectricChargingStations[diLPForGVL,diCounterForGVL].rTargetPowerEMS := 0;	
		END_FOR
		
			//Counter for ECS
			diCounterForGVL := diCounterForGVL + 1;
				diCounterForGVL := LIMIT(0,diCounterForGVL,Constants_Energy.diMaxNumberOfElectricChargingStations);
					//Back to the init step
					IF diCounterForGVL >= Constants_Energy.diMaxNumberOfElectricChargingStations THEN iStateGVLData := 0; END_IF

	10://Clear old Data on GVL 		
		Lynus_Standards.GVL_Energy.stDataElectricChargingStations[diNrOfEMS_IN_CP,diNrOfECS_OUT].bEnabled := FALSE;
			Lynus_Standards.GVL_Energy.stDataElectricChargingStations[diNrOfEMS_IN_CP,diNrOfECS_OUT].bIsControllable := FALSE;
				Lynus_Standards.GVL_Energy.stDataElectricChargingStations[diNrOfEMS_IN_CP,diNrOfECS_OUT].byErrorWarning := 0;
					Lynus_Standards.GVL_Energy.stDataElectricChargingStations[diNrOfEMS_IN_CP,diNrOfECS_OUT].byPriority := 0;
						Lynus_Standards.GVL_Energy.stDataElectricChargingStations[diNrOfEMS_IN_CP,diNrOfECS_OUT].lrPower := 0;
							Lynus_Standards.GVL_Energy.stDataElectricChargingStations[diNrOfEMS_IN_CP,diNrOfECS_OUT].lrPowerConsumption := 0;
								Lynus_Standards.GVL_Energy.stDataElectricChargingStations[diNrOfEMS_IN_CP,diNrOfECS_OUT].lrPowerProduction := 0;
									Lynus_Standards.GVL_Energy.stDataElectricChargingStations[diNrOfEMS_IN_CP,diNrOfECS_OUT].rMaxPower := 0;
										Lynus_Standards.GVL_Energy.stDataElectricChargingStations[diNrOfEMS_IN_CP,diNrOfECS_OUT].byElectricFuseLine := 0;
									
		diNrOfEMS_IN_CP := diNrOfEMS_IN;
			//Back to the init step
			iStateGVLData := 0;

END_CASE 	 

IF diNrOfECS_OUT > 0 AND fbNumberDevice.bNumberIsCalculatet AND diNrOfEMS_IN > 0 THEN
	Lynus_Standards.GVL_Energy.stDataElectricChargingStations[diNrOfEMS_IN,diNrOfECS_OUT].bEnabled := fbCS.stDataECSOut.bEnabled;
		Lynus_Standards.GVL_Energy.stDataElectricChargingStations[diNrOfEMS_IN,diNrOfECS_OUT].bIsControllable := TRUE;
			Lynus_Standards.GVL_Energy.stDataElectricChargingStations[diNrOfEMS_IN,diNrOfECS_OUT].byErrorWarning := fbCS.stDataECSOut.byErrorWarning;
				Lynus_Standards.GVL_Energy.stDataElectricChargingStations[diNrOfEMS_IN,diNrOfECS_OUT].byPriority := fbCS.stDataECSOut.byPriority;
					Lynus_Standards.GVL_Energy.stDataElectricChargingStations[diNrOfEMS_IN,diNrOfECS_OUT].lrPower := fbCS.stDataECSOut.lrTotalPower;
						Lynus_Standards.GVL_Energy.stDataElectricChargingStations[diNrOfEMS_IN,diNrOfECS_OUT].lrPowerConsumption := fbCS.stDataECSOut.lrTotalPowerConsumption;
							Lynus_Standards.GVL_Energy.stDataElectricChargingStations[diNrOfEMS_IN,diNrOfECS_OUT].lrPowerProduction := fbCS.stDataECSOut.lrTotalPowerProduction;
								Lynus_Standards.GVL_Energy.stDataElectricChargingStations[diNrOfEMS_IN,diNrOfECS_OUT].rMaxPower := fbCS.stDataECSOut.rMaxPower;	
									Lynus_Standards.GVL_Energy.stDataElectricChargingStations[diNrOfEMS_IN,diNrOfECS_OUT].byElectricFuseLine := byElectricFuseLine;
END_IF 

(*----------------------------------------------------------Save persistent data----------------------------------------------------------------*)

arrPD[1](lrValue:= BOOL_TO_LREAL(bEnable), bEventBasedActive=> );
arrPD[2](lrValue:= BOOL_TO_LREAL(bPowerDataInvers), bEventBasedActive=> );
arrPD[3](lrValue:= DINT_TO_LREAL(diNrOfEMS_IN), bEventBasedActive=> );
arrPD[4](lrValue:= DINT_TO_LREAL(diNrOfEM_IN_CS), bEventBasedActive=> );
arrPD[5](lrValue:= BOOL_TO_LREAL(stSetupECS.bManualyOn), bEventBasedActive=> );
arrPD[6](lrValue:= BOOL_TO_LREAL(stSetupECS.bOnEmergPowerOff), bEventBasedActive=> );
arrPD[7](lrValue:= BYTE_TO_LREAL(stSetupECS.byCSMinPower), bEventBasedActive=> );
arrPD[8](lrValue:= BYTE_TO_LREAL(stSetupECS.byDisableSOC), bEventBasedActive=> );
arrPD[9](lrValue:= BYTE_TO_LREAL(stSetupECS.byEnableSOC), bEventBasedActive=> );
arrPD[10](lrValue:= BYTE_TO_LREAL(stSetupECS.byManualyTargetPower), bEventBasedActive=> );
arrPD[11](lrValue:= BYTE_TO_LREAL(stSetupECS.byPriority), bEventBasedActive=> );
arrPD[12](lrValue:= REAL_TO_LREAL(stSetupECS.rMaxPower), bEventBasedActive=> );
arrPD[13](lrValue:= DINT_TO_LREAL(diNrOfEMS_IN_CP), bEventBasedActive=> );
arrPD[14](lrValue:= BYTE_TO_LREAL(byElectricFuseLine), bEventBasedActive=> );
arrPD[15](lrValue:= UINT_TO_LREAL(uiFailsafeCurrent), bEventBasedActive=> );
arrPD[16](lrValue:= UINT_TO_LREAL(uiFailsafeTimeOut), bEventBasedActive=> );
fbPDString(sText:= sIPAdress, bEventBasedActive=> );

END_FUNCTION_BLOCK

// ---- POUs/prgEM.TcPOU
PROGRAM prgEM
VAR
	fbKBusState		: FB_K_Bus_State;
	fbEM1			: FB_EM_Beckhoff_KL3403;

	bEnable: BOOL:=TRUE;
	lrPowerKeba: LREAL;				//{#lynus.ag#()}
	lrCounterKeba: LREAL;			//{#lynus.ag#()}
	lrPowerKeba_1: LREAL;			//{#lynus.ag#()}
	lrPowerKeba_2: LREAL;			//{#lynus.ag#()}
	lrPowerKeba_3: LREAL;			//{#lynus.ag#()}
	lrVoltageKeba_1: LREAL;			//{#lynus.ag#()}
	lrVoltageKeba_2: LREAL;			//{#lynus.ag#()}
	lrVoltageKeba_3: LREAL;			//{#lynus.ag#()}
	lrCurrentKeba_1: LREAL;			//{#lynus.ag#()}
	lrCurrentKeba_2: LREAL;			//{#lynus.ag#()}
	lrCurrentKeba_3: LREAL;			//{#lynus.ag#()}
	lrEnergyKeba: LREAL;			//{#lynus.ag#()}
END_VAR


fbKBusState(	uiKBusState_OUT=> , 
				b_Kbus_notOk=> , 
				word_ErrorCount=> );
//The mapping OF THIS FUNCTION must be linked with the KL3403 in the E/A Part
// KEBA CS
fbEM1(
	bEnable:= bEnable, 
	bChannel1Invers:= FALSE,				//Invert power data when transformer are mounted upside down
	bChannel2Invers:= FALSE,			
	bChannel3Invers:= FALSE,
	uiCurrentTransformerRatioL1:= 400, //Transformer ratio on the secondary side
	uiCurrentTransformerRatioL2:= 400, 
	uiCurrentTransformerRatioL3:= 400, 
	uiKBusState_IN:= fbKBusState.uiKBusState_OUT, 
	stDataEMPower=> , 
	stDataEMCounter=> , 
	stDataEMPowerRealTime=> , 
	stDataEMCounterRealTime=> , 
	diNrOfEM_OUT=> );
	
lrPowerKeba := fbEM1.stDataEMPower.lrPowerTotal;
lrCounterKeba := fbEM1.stDataEMCounter.lrTotalCounterEnergy_Consumption;	
lrPowerKeba_1 := fbEM1.stDataEMPower.lrPowerL1;
lrPowerKeba_2 := fbEM1.stDataEMPower.lrPowerL2;
lrPowerKeba_3 := fbEM1.stDataEMPower.lrPowerL3;
lrVoltageKeba_1 := fbEM1.stDataEMPower.lrVoltageL1N;
lrVoltageKeba_2 := fbEM1.stDataEMPower.lrVoltageL2N;
lrVoltageKeba_3 := fbEM1.stDataEMPower.lrVoltageL3N;
lrCurrentKeba_1 := fbEM1.stDataEMPower.lrCurrentL1;
lrCurrentKeba_2 := fbEM1.stDataEMPower.lrCurrentL2;
lrCurrentKeba_3 := fbEM1.stDataEMPower.lrCurrentL3;
lrEnergyKeba	:= fbEM1.stDataEMCounter.lrTotalCounterEnergy_Consumption;

END_PROGRAM

// ---- POUs/prgPersistent.TcPOU
PROGRAM prgPersistent
VAR
	fbUSV		: FB_WritePersistentData_CX81xx;
	fb_Reboot: NT_Reboot;
	mTest: BOOL;
	ton_liveCount: Ton;
	int_LiveCount: INT;										//{#lynus.ag#()}
END_VAR

fbUSV(
	eSaveModeData:= eUSVSaveMode.eSaveWhenPowerfail, 
	bLoadPersistentDataOk=> , 
	bPowerFailDetect=> , 
	bError=> , 
	bySaveProcess=> , 
	dwStorageLast24h=> , 
	udiErrorCode=> );
	
fb_Reboot (
	netid := '',
	delay := 5,
	start := mTest);
	

ton_liveCount( 	IN := NOT ton_liveCount.Q,
				PT := T#1M);
				
IF ton_liveCount.Q THEN
	int_LiveCount := int_LiveCount+1;	
END_IF

END_PROGRAM

// ---- POUs/prgMain.TcPOU
PROGRAM prgMain
VAR
	int_Temp_1_1 	AT%I*	: INT;
	int_Temp_1_2 	AT%I*	: INT;
	int_Temp_1_3 	AT%I*	: INT;
	int_Temp_1_4 	AT%I*	: INT;
	int_Temp_2_1 	AT%I*	: INT;
	int_Temp_2_2 	AT%I*	: INT;
	int_Temp_2_3 	AT%I*	: INT;
	int_Temp_2_4 	AT%I*	: INT;	
	real_Temp_K1			: REAL;											//{#lynus.ag#()}
	real_Temp_K2			: REAL;											//{#lynus.ag#()}
	real_Temp_W11			: REAL;											//{#lynus.ag#()}
	real_Temp_W12			: REAL;											//{#lynus.ag#()}
	real_Temp_W21			: REAL;											//{#lynus.ag#()}
	real_Temp_W22			: REAL;											//{#lynus.ag#()}
	real_Temp_WZ			: REAL;											//{#lynus.ag#()}
// Kanal 2.2
	fb_Config_22			: FB_KL320xConfig;
	stInData_22   AT%I*		: ST_KL320xInData;
	stOutData_22  AT%Q*		: ST_KL320xOutData;
// Kanal 2.4
	fb_Config_24			: FB_KL320xConfig;
	stInData_24   AT%I*		: ST_KL320xInData;
	stOutData_24  AT%Q*		: ST_KL320xOutData;
	fb_curve				: fb_CurveRead;
	fb_curve2				: fb_CurveRead;
// Kanal W22
	fb_Config_W22			: FB_KL320xConfig;
	stInData_W22   AT%I*		: ST_KL320xInData;
	stOutData_W22  AT%Q*		: ST_KL320xOutData;
	mTest:BOOL;
	
	real_Temp_Outside: REAL;												//{#lynus.ag#()}
	fbShelly1					: FB_Shelly_Pro4PM;
	fbShelly2					: FB_Shelly_Pro2pm;
	bPro4pmCH1_on				: BOOL;											//{#lynus.ag#()}
	bPro4pmCH2_on				: BOOL;											//{#lynus.ag#()}
	bPro4pmCH3_on				: BOOL;											//{#lynus.ag#()}
	bPro4pmCH4_on				: BOOL;											//{#lynus.ag#()}
	bPro2pmCH1_on				: BOOL;											//{#lynus.ag#()}
	bPro2pmCH2_on				: BOOL;											//{#lynus.ag#()}
	
	int_liveCount: INT;
	


	int_Temp_W2_2: INT;
	fb_curveW22				: fb_CurveRead;

END_VAR
VAR PERSISTENT
	int_Offset_W22: INT;														//{#lynus.ag#()}
	int_Offset_Outside: INT;													//{#lynus.ag#()}

END_VAR

int_liveCount := int_liveCount +1;


real_Temp_K1 	:= INT_TO_REAL(int_Temp_1_1)/10;
real_Temp_K2 	:= INT_TO_REAL(int_Temp_1_3)/10;
real_Temp_W11 	:= INT_TO_REAL(int_Temp_1_2)/10;
real_Temp_W12 	:= INT_TO_REAL(int_Temp_1_4)/10;
real_Temp_W21 	:= INT_TO_REAL(int_Temp_2_1)/10;
real_Temp_W22 	:= INT_TO_REAL(REAL_TO_INT(fb_curveW22.real_y*10))/10;
real_Temp_WZ	:= INT_TO_REAL(REAL_TO_INT(fb_curve.real_y*10))/10;
real_Temp_Outside := INT_TO_REAL(REAL_TO_INT(fb_curve2.real_y*10))/10;

int_Temp_2_2 := stInData_22.iDataIn;
int_Temp_2_4 := stInData_24.iDataIn;
int_Temp_W2_2 := stInData_W22.iDataIn;

fb_Config_22(
	bConfigurate:= , 
	bReadConfig:= , 
	iSetSensorType:= , 
	tTimeout:= , 
	bBusy=> , 
	bError=> , 
	iErrorId=> , 
	iState=> , 
	iDataIn=> , 
	iTerminalType=> , 
	iSpecialType=> , 
	iFirmwareVersion=> , 
	sDescription=> , 
	sSensorType=> , 
	bTwoWiredConnection=> , 
	stInData:= stInData_22 , 
	stOutData:= stOutData_22);
	
fb_Config_24(
	bConfigurate:= , 
	bReadConfig:= , 
	iSetSensorType:= , 
	tTimeout:= , 
	bBusy=> , 
	bError=> , 
	iErrorId=> , 
	iState=> , 
	iDataIn=> , 
	iTerminalType=> , 
	iSpecialType=> , 
	iFirmwareVersion=> , 
	sDescription=> , 
	sSensorType=> , 
	bTwoWiredConnection=> , 
	stInData:= stInData_24, 
	stOutData:= stOutData_24);

fb_Config_W22(
	bConfigurate:= , 
	bReadConfig:= , 
	iSetSensorType:= , 
	tTimeout:= , 
	bBusy=> , 
	bError=> , 
	iErrorId=> , 
	iState=> , 
	iDataIn=> , 
	iTerminalType=> , 
	iSpecialType=> , 
	iFirmwareVersion=> , 
	sDescription=> , 
	sSensorType=> , 
	bTwoWiredConnection=> , 
	stInData:= stInData_W22 , 
	stOutData:= stOutData_W22);	
	
// interpolation NTC 1.8k zwischen 10°C - 40°C
fb_curve(
	real_x:= (INT_TO_REAL(int_Temp_2_4)/2) , 
	real_x1:= 1040, 
	real_y1:= 40, 
	real_x2:= 1480, 
	real_y2:= 30, 
	real_x3:= 2200 , 
	real_y3:= 20, 
	real_x4:= 3330 , 
	real_y4:= 10, 
	real_y=> , 
	m_x_Outside=> );
	
// interpolation PT100 mit 6,5Ohm Leitungswiederstand zwischen -20°C und +40°C
fb_curve2(
	real_x:= (INT_TO_REAL(int_Temp_2_2))/10-int_Offset_Outside , 
	real_x1:= 92, 
	real_y1:= -20, 
	real_x2:= 100, 
	real_y2:= 0, 
	real_x3:= 107.79 , 
	real_y3:= 20, 
	real_x4:= 115.54 , 
	real_y4:= 40, 
	real_y=> , 
	m_x_Outside=> );


// interpolation PT100 mit 10Ohm Leitungswiederstand zwischen -20°C und +40°C
fb_curveW22(
	real_x:= (INT_TO_REAL(int_Temp_W2_2))/10-int_Offset_W22 , 
	real_x1:= 92, 
	real_y1:= -20, 
	real_x2:= 100, 
	real_y2:= 0, 
	real_x3:= 107.79 , 
	real_y3:= 20, 
	real_x4:= 115.54 , 
	real_y4:= 40, 
	real_y=> , 
	m_x_Outside=> );	
	// Shelly pro 4 pm
	
fbShelly1(
	bStart:= TRUE, 
	tDelayRequest:= T#3S, 
	sHostname:= '192.168.1.20', 
	bValidResult=> , 
	bBusy=> , 
	bError=> , 
	bDone=> , 
	hrErrorCode=> ,
	lrpowerP1=> , 
	lrvoltageP1=> , 
	lrenergyP1=> ,
	lrpowerP2=> , 
	lrvoltageP2=> , 
	lrenergyP2=> ,
	bOnP1:= bPro4pmCH1_on,
	bOffP1:= NOT bPro4pmCH1_on ,
	bStateP1=> ,
	bOnP2:= bPro4pmCH2_on ,
	bOffP2:= NOT bPro4pmCH2_on ,
	bStateP2=> ,
	bOnP3:= bPro4pmCH3_on ,
	bOffP3:= NOT bPro4pmCH3_on ,
	bStateP3=>  ,
	bOnP4:= bPro4pmCH4_on ,
	bOffP4:= NOT bPro4pmCH4_on ,
	bStateP4=>  );	
// shelly pr 2pm

fbShelly2(
	bStart:= TRUE , 
	tDelayRequest:= T#3S, 
	sHostname:= '192.168.1.21', 
	bOnP1:= bPro2pmCH1_on, 
	bOffP1:= NOT bPro2pmCH1_on, 
	bOnP2:= bPro2pmCH2_on , 
	bOffP2:= not bPro2pmCH2_on, 
	bValidResult=> , 
	bBusy=> , 
	bError=> , 
	bDone=> , 
	bConnected=> , 
	hrErrorCode=> , 
	lrpowerP1=> , 
	lrvoltageP1=> , 
	lrenergyP1=> , 
	lrpowerP2=> , 
	lrvoltageP2=> , 
	lrenergyP2=> , 
	bStateP1=> , 
	bStateP2=> );

END_PROGRAM

// ---- POUs/FB_CurveRead.TcPOU
FUNCTION_BLOCK FB_CurveRead
VAR_INPUT
	real_x	:REAL;
	real_x1	:REAL;
	real_y1	:REAL;
	real_x2	:REAL;
	real_y2	:REAL;
	real_x3	:REAL;
	real_y3	:REAL;
	real_x4	:REAL;
	real_y4	:REAL;
END_VAR
VAR_OUTPUT
	real_y	:REAL;
	m_x_Outside: BOOL;
END_VAR
VAR
END_VAR

IF real_x<real_x1 THEN
	m_x_Outside:=TRUE;
	real_y:=real_y1;
ELSIF real_x>real_x4 THEN
	m_x_Outside:=TRUE;
	real_y:=real_y4;
ELSIF real_x>=real_x1 AND real_x<real_x2 AND (real_x2-real_x1)<>0 THEN
	m_x_Outside:=FALSE;
	real_y:=(real_y2-real_y1)/(real_x2-real_x1)*(real_x-real_x1)+real_y1;
ELSIF real_x>=real_x2 AND real_x<real_x3 AND (real_x3-real_x2)<>0 THEN
	m_x_Outside:=FALSE;
	real_y:=(real_y3-real_y2)/(real_x3-real_x2)*(real_x-real_x2)+real_y2;
ELSIF real_x>=real_x3 AND real_x<=real_x4 AND (real_x4-real_x3)<>0 THEN
	m_x_Outside:=FALSE;
	real_y:=(real_y4-real_y3)/(real_x4-real_x3)*(real_x-real_x3)+real_y3;
END_IF

END_FUNCTION_BLOCK

// ---- FBs/FB_Shelly_Pro4PM.TcPOU
FUNCTION_BLOCK FB_Shelly_Pro4PM
VAR_INPUT
	bStart				: BOOL;
	tDelayRequest		: TIME := T#3S;		//Timer for delay before start with the next read or write Request
	sHostname			: STRING(255);		//Hostname or IP Adress from the Server
	bOnP1				: BOOL;
	bOffP1				: BOOL;
	bOnP2				: BOOL;
	bOffP2				: BOOL;
	bOnP3				: BOOL;
	bOffP3				: BOOL;
	bOnP4				: BOOL;
	bOffP4				: BOOL;
END_VAR

VAR_IN_OUT
END_VAR

VAR_OUTPUT
	bValidResult				: BOOL;															//Valid Result received from Server
    bBusy						: BOOL;															//Function is Busy
    bError						: BOOL;															//Error sucess
	bDone						: BOOL;															//True after the decoding from the received Json File
	bConnected					: BOOL;															//Connection to the Server
	lrpowerP1					: LREAL;														//Received Value
	lrvoltageP1					: LREAL;														//Received Value
	lrenergyP1					: LREAL;														//Received Value
	lrpowerP2					: LREAL;														//Received Value
	lrvoltageP2					: LREAL;														//Received Value
	lrenergyP2					: LREAL;
	lrpowerP3					: LREAL;														//Received Value
	lrvoltageP3					: LREAL;														//Received Value
	lrenergyP3					: LREAL;
	lrpowerP4					: LREAL;														//Received Value
	lrvoltageP4					: LREAL;														//Received Value
	lrenergyP4					: LREAL;	
	hrErrorCode       			: HRESULT;														//Error Result from Http Client
	bStateP1					: BOOL;
	bStateP2					: BOOL;
	bStateP3					: BOOL;
	bStateP4					: BOOL;
END_VAR

VAR
	fbClient					: FB_IotHttpClient;
	fbHttpGet					: FB_Shelly_Pro4PM_Helper;
	timStartRequest				: TON;															//Timer to Start the Request
	FPStartRequest				: R_TRIG;														//Internal positive Edge
	FPDone						: R_TRIG;														//Internal positive Edge
	FNStart						: F_TRIG;														//Internal negative Edge
	SwitchOnP1					: R_TRIG;
	SwitchOffP1					: R_TRIG;
	SwitchOnP2					: R_TRIG;
	SwitchOffP2					: R_TRIG;
	SwitchOnP3					: R_TRIG;
	SwitchOffP3					: R_TRIG;
	SwitchOnP4					: R_TRIG;
	SwitchOffP4					: R_TRIG;
END_VAR

(*------------------------------------------------------------------------------------Configure HTTP Client------------------------------------------------------------------------------------------------------*)

fbClient.sHostName := sHostname;
fbClient.tConnectionTimeout := tDelayRequest;

IF NOT fbClient.bConfigured THEN 
	fbClient.nHostPort:= 80;
	fbClient.bKeepAlive := TRUE;
	fbClient.tConnectionTimeout := T#2S;
END_IF


//Timer to start the Request
FPStartRequest(CLK:= bStart, Q=> );
	timStartRequest(IN:= fbClient.bConfigured AND bStart AND NOT timStartRequest.Q, PT:= tDelayRequest, Q=> , ET=> );
		IF ((timStartRequest.Q AND NOT bBusy) OR (FPStartRequest.Q AND NOT bBusy AND fbClient.bConfigured)) THEN fbHttpGet.bSend := TRUE; END_IF

				
//Http Get Function
fbHttpGet(
	lrapowerP1 => lrpowerP1, 
	lrvoltageP1 => lrvoltageP1, 
	lraenergyP1 => lrenergyP1,
	lrapowerP2 => lrpowerP2, 
	lrvoltageP2 => lrvoltageP2, 
	lraenergyP2 => lrenergyP2,
	lrapowerP3 => lrpowerP3, 
	lrvoltageP3 => lrvoltageP3, 
	lraenergyP3 => lrenergyP3,
	lrapowerP4 => lrpowerP4, 
	lrvoltageP4 => lrvoltageP4, 
	lraenergyP4 => lrenergyP4, 
	bSend:= , 
	fbClient:= fbClient, 
	bBusy=> bBusy, 
	bError=> ,
	sContentS0=> ,
	sContentS1=> ,
	sContentS2=> ,
	sContentS3=> ,
	bStateP1=>bStateP1,
	bStateP2=>bStateP2,
	bStateP3=>bStateP3,
	bStateP4=>bStateP4 );


fbHttpGet.bSend := FALSE;

FPDone(CLK:= bDone, Q=> );

(*
//Http Client
FNStart(CLK:= bStart, Q=> );
	IF FNStart.Q THEN fbClient.Disconnect(); END_IF
*)

fbClient.Execute();

//Error
IF fbHttpGet.bError OR fbClient.bError THEN bError := TRUE; ELSE bError := FALSE; END_IF	
	hrErrorCode := fbClient.hrErrorCode;
	

// Relay Control, Switch P1
SwitchOnP1(CLK:=bOnP1);
IF SwitchOnP1.Q THEN
	fbHttpGet.bSetOnP1 := TRUE;
END_IF

SwitchOffP1(CLK:=bOffP1);
IF SwitchOffP1.Q THEN
	fbHttpGet.bSetOffP1 := TRUE;
END_IF

// Relay Control, Switch P2
SwitchOnP2(CLK:=bOnP2);
IF SwitchOnP2.Q THEN
	fbHttpGet.bSetOnP2 := TRUE;
END_IF

SwitchOffP2(CLK:=bOffP2);
IF SwitchOffP2.Q THEN
	fbHttpGet.bSetOffP2 := TRUE;
END_IF

// Relay Control, Switch P3
SwitchOnP3(CLK:=bOnP3);
IF SwitchOnP3.Q THEN
	fbHttpGet.bSetOnP3 := TRUE;
END_IF

SwitchOffP3(CLK:=bOffP3);
IF SwitchOffP3.Q THEN
	fbHttpGet.bSetOffP3 := TRUE;
END_IF

// Relay Control, Switch P4
SwitchOnP4(CLK:=bOnP4);
IF SwitchOnP4.Q THEN
	fbHttpGet.bSetOnP4 := TRUE;
END_IF

SwitchOffP4(CLK:=bOffP4);
IF SwitchOffP4.Q THEN
	fbHttpGet.bSetOffP4 := TRUE;
END_IF

END_FUNCTION_BLOCK

// ---- FBs/FB_Shelly_Pro4PM_Helper.TcPOU
FUNCTION_BLOCK FB_Shelly_Pro4PM_Helper
VAR_INPUT
	bSend			: BOOL;
	bSetOnP1		: BOOL;
	bSetOffP1		: BOOL;
	bSetOnP2		: BOOL;
	bSetOffP2		: BOOL;
	bSetOnP3		: BOOL;
	bSetOffP3		: BOOL;
	bSetOnP4		: BOOL;
	bSetOffP4		: BOOL;
END_VAR

VAR_IN_OUT
	fbClient		: FB_IotHttpClient;
END_VAR

VAR_OUTPUT
	bBusy			: BOOL;
	bError			: BOOL;
	bStateP1		: BOOL;
	bStateP2		: BOOL;
	bStateP3		: BOOL;
	bStateP4		: BOOL;
	lrapowerP1		: LREAL;
	lrvoltageP1		: LREAL;
	lraenergyP1		: LREAL;
	lrapowerP2		: LREAL;
	lrvoltageP2		: LREAL;
	lraenergyP2		: LREAL;
	lrapowerP3		: LREAL;
	lrvoltageP3		: LREAL;
	lraenergyP3		: LREAL;
	lrapowerP4		: LREAL;
	lrvoltageP4		: LREAL;
	lraenergyP4		: LREAL;
END_VAR

VAR
	fbRequestSwitch0	: FB_IotHttpRequest;
	fbRequestSwitch1	: FB_IotHttpRequest;
	fbRequestSwitch2	: FB_IotHttpRequest;
	fbRequestSwitch3	: FB_IotHttpRequest;
	fbJson				: FB_JsonDomParser;
	nState				: UDINT;
	RisingEdge			: R_TRIG;
	RisingEdgeSetOnP1	: R_TRIG;
	RisingEdgeSetOffP1	: R_TRIG;
	RisingEdgeSetOnP2	: R_TRIG;
	RisingEdgeSetOffP2	: R_TRIG;
	RisingEdgeSetOnP3	: R_TRIG;
	RisingEdgeSetOffP3	: R_TRIG;
	RisingEdgeSetOnP4	: R_TRIG;
	RisingEdgeSetOffP4	: R_TRIG;
	timTimeout			: TON;
	tTimeOut			: TIME := T#30S;
	timTimeoutSwitch	: TON;
	tTimeOutSwitch		: TIME := T#5S;
	
	bGetContentResult	: BOOL;
	sContentS0			: STRING(511);
	sContentS1			: STRING(511);
	sContentS2			: STRING(511);
	sContentS3			: STRING(511);
	
	bGetJsonResult		: BOOL;
	jsonDoc				: SJsonValue;
	jsonVal				: SJsonValue;
	
	nReqCount			: UDINT;	
	nResCount			: UDINT;
	nValidResCount		: UDINT;
	nErrCount			: UDINT;
END_VAR

//Timer for Timeout
timTimeout(IN:= nState = 1 AND bBusy, PT:= tTimeOut, Q=> , ET=> );
	IF timTimeout.Q THEN 
		nState := 0;
		bBusy := FALSE;
	END_IF
	
timTimeoutSwitch(IN:= bSetOnP1 OR bSetOffP1 OR bSetOnP2 OR bSetOffP2 OR bSetOnP3 OR bSetOffP3 OR bSetOnP4 OR bSetOffP4, PT:= tTimeOut, Q=> , ET=> );
	IF timTimeoutSwitch.Q THEN 
		bSetOnP1 := FALSE;
		bSetOffP1 := FALSE;
		bSetOnP2 := FALSE;
		bSetOffP2 := FALSE;
		bSetOnP3 := FALSE;
		bSetOffP3 := FALSE;
		bSetOnP4 := FALSE;
		bSetOffP4 := FALSE;
	END_IF

RisingEdge(CLK:= bSend );
RisingEdgeSetOnP1(CLK:= bSetOnP1 );
RisingEdgeSetOffP1(CLK:= bSetOffP1 );
RisingEdgeSetOnP2(CLK:= bSetOnP2 );
RisingEdgeSetOffP2(CLK:= bSetOffP2 );
RisingEdgeSetOnP3(CLK:= bSetOnP3 );
RisingEdgeSetOffP3(CLK:= bSetOffP3 );
RisingEdgeSetOnP4(CLK:= bSetOnP4 );
RisingEdgeSetOffP4(CLK:= bSetOffP4 );

CASE nState OF
0:	
	IF RisingEdge.Q THEN 
		IF
			fbRequestSwitch0.SendRequest(sUri:='/rpc/Switch.GetStatus?id=0', fbClient:=fbClient, eRequestType:=ETcIotHttpRequestType.HTTP_Get, 0, 0, 0) AND
			fbRequestSwitch1.SendRequest(sUri:='/rpc/Switch.GetStatus?id=1', fbClient:=fbClient, eRequestType:=ETcIotHttpRequestType.HTTP_Get, 0, 0, 0) AND
			fbRequestSwitch2.SendRequest(sUri:='/rpc/Switch.GetStatus?id=2', fbClient:=fbClient, eRequestType:=ETcIotHttpRequestType.HTTP_Get, 0, 0, 0) AND
			fbRequestSwitch3.SendRequest(sUri:='/rpc/Switch.GetStatus?id=3', fbClient:=fbClient, eRequestType:=ETcIotHttpRequestType.HTTP_Get, 0, 0, 0) THEN				
			nState:= 1;
			nReqCount:= nReqCount+1;
			bBusy:= TRUE;
			bError:= FALSE;
		END_IF					
	END_IF
	
	IF RisingEdgeSetOnP1.Q THEN 
		IF
			fbRequestSwitch0.SendRequest(sUri:='/rpc/Switch.Set?id=0&on=true', fbClient:=fbClient, eRequestType:=ETcIotHttpRequestType.HTTP_Get, 0, 0, 0) THEN				
			bSetOnP1 := FALSE;
			nState:= 1;
			bBusy:= TRUE;
			bError:= FALSE;
		END_IF					
	END_IF
	
	IF RisingEdgeSetOffP1.Q THEN 
		IF
			fbRequestSwitch0.SendRequest(sUri:='/rpc/Switch.Set?id=0&on=false', fbClient:=fbClient, eRequestType:=ETcIotHttpRequestType.HTTP_Get, 0, 0, 0) THEN				
			bSetOffP1 := FALSE;
			nState:= 1;
			bBusy:= TRUE;
			bError:= FALSE;
		END_IF					
	END_IF
	
	IF RisingEdgeSetOnP2.Q THEN 
		IF
			fbRequestSwitch1.SendRequest(sUri:='/rpc/Switch.Set?id=1&on=true', fbClient:=fbClient, eRequestType:=ETcIotHttpRequestType.HTTP_Get, 0, 0, 0) THEN				
			bSetOnP2 := FALSE;
			nState:= 1;
			bBusy:= TRUE;
			bError:= FALSE;
		END_IF					
	END_IF
	
	IF RisingEdgeSetOffP2.Q THEN 
		IF
			fbRequestSwitch1.SendRequest(sUri:='/rpc/Switch.Set?id=1&on=false', fbClient:=fbClient, eRequestType:=ETcIotHttpRequestType.HTTP_Get, 0, 0, 0) THEN				
			bSetOffP2 := FALSE;
			nState:= 1;
			bBusy:= TRUE;
			bError:= FALSE;
		END_IF					
	END_IF
	
	IF RisingEdgeSetOnP3.Q THEN 
		IF
			fbRequestSwitch2.SendRequest(sUri:='/rpc/Switch.Set?id=2&on=true', fbClient:=fbClient, eRequestType:=ETcIotHttpRequestType.HTTP_Get, 0, 0, 0) THEN				
			bSetOnP3 := FALSE;
			nState:= 1;
			bBusy:= TRUE;
			bError:= FALSE;
		END_IF					
	END_IF
	
	IF RisingEdgeSetOffP3.Q THEN 
		IF
			fbRequestSwitch2.SendRequest(sUri:='/rpc/Switch.Set?id=2&on=false', fbClient:=fbClient, eRequestType:=ETcIotHttpRequestType.HTTP_Get, 0, 0, 0) THEN				
			bSetOffP3 := FALSE;
			nState:= 1;
			bBusy:= TRUE;
			bError:= FALSE;
		END_IF					
	END_IF
	
	IF RisingEdgeSetOnP4.Q THEN 
		IF
			fbRequestSwitch3.SendRequest(sUri:='/rpc/Switch.Set?id=3&on=true', fbClient:=fbClient, eRequestType:=ETcIotHttpRequestType.HTTP_Get, 0, 0, 0) THEN				
			bSetOnP4 := FALSE;
			nState:= 1;
			bBusy:= TRUE;
			bError:= FALSE;
		END_IF					
	END_IF
	
	IF RisingEdgeSetOffP4.Q THEN 
		IF
			fbRequestSwitch3.SendRequest(sUri:='/rpc/Switch.Set?id=3&on=false', fbClient:=fbClient, eRequestType:=ETcIotHttpRequestType.HTTP_Get, 0, 0, 0) THEN				
			bSetOffP4 := FALSE;
			nState:= 1;
			bBusy:= TRUE;
			bError:= FALSE;
		END_IF					
	END_IF
	
1:
	IF NOT fbRequestSwitch0.bBusy AND NOT fbRequestSwitch1.bBusy AND NOT fbRequestSwitch2.bBusy AND NOT fbRequestSwitch3.bBusy THEN
		bError:= TRUE;
		
		IF NOT fbRequestSwitch0.bError THEN				 
			bGetContentResult:= fbRequestSwitch0.GetContent(pContent:= ADR(sContentS0), nContentSize:= SIZEOF(sContentS0), bSetNullTermination:= TRUE);
			IF fbRequestSwitch0.nStatusCode >= 200 AND fbRequestSwitch0.nStatusCode < 300 THEN
				bGetJsonResult:= FALSE;
				jsonDoc:= fbRequestSwitch0.GetJsonDomContent(fbJson);
				IF jsonDoc <> 0 THEN
					bGetJsonResult:= TRUE;
					IF fbJson.HasMember(jsonDoc, 'output')  THEN
						jsonVal:= fbJson.FindMember(jsonDoc, 'output');
						nValidResCount:= nValidResCount+1;					
						IF fbJson.IsBool(jsonVal) THEN							
							bStateP1:= fbJson.GetBool(jsonVal);									
						END_IF
						jsonVal:= fbJson.FindMember(jsonDoc, 'apower');
						nValidResCount:= nValidResCount+1;
						IF fbJson.IsDouble(jsonVal) THEN							
							lrapowerP1:= fbJson.GetDouble(jsonVal);									
						END_IF
						jsonVal:= fbJson.FindMember(jsonDoc, 'voltage');
						nValidResCount:= nValidResCount+1;					
						IF fbJson.IsDouble(jsonVal) THEN							
							lrvoltageP1:= fbJson.GetDouble(jsonVal);									
						END_IF
						jsonVal:= fbJson.FindMember(jsonDoc, 'aenergy');
                        IF fbJson.HasMember(jsonVal, 'total') THEN
                            jsonVal:= fbJson.FindMember(jsonVal, 'total');
                            nValidResCount:= nValidResCount+1;
                            IF fbJson.IsDouble(jsonVal) THEN
                                lraenergyP1:= fbJson.GetDouble(jsonVal);
                            END_IF
						bError:= FALSE;
						END_IF
					END_IF						
				nResCount:= nResCount+1;			
				END_IF
			END_IF
		END_IF
		
		IF NOT fbRequestSwitch1.bError THEN				 
			bGetContentResult:= fbRequestSwitch1.GetContent(pContent:= ADR(sContentS1), nContentSize:= SIZEOF(sContentS1), bSetNullTermination:= TRUE);
			IF fbRequestSwitch1.nStatusCode >= 200 AND fbRequestSwitch1.nStatusCode < 300 THEN
				bGetJsonResult:= FALSE;
				jsonDoc:= fbRequestSwitch1.GetJsonDomContent(fbJson);
				IF jsonDoc <> 0 THEN
					bGetJsonResult:= TRUE;
					IF fbJson.HasMember(jsonDoc, 'output')  THEN
						jsonVal:= fbJson.FindMember(jsonDoc, 'output');
						nValidResCount:= nValidResCount+1;					
						IF fbJson.IsBool(jsonVal) THEN							
							bStateP2:= fbJson.GetBool(jsonVal);									
						END_IF
						jsonVal:= fbJson.FindMember(jsonDoc, 'apower');
						nValidResCount:= nValidResCount+1;
						IF fbJson.IsDouble(jsonVal) THEN							
							lrapowerP2:= fbJson.GetDouble(jsonVal);									
						END_IF
						jsonVal:= fbJson.FindMember(jsonDoc, 'voltage');
						nValidResCount:= nValidResCount+1;					
						IF fbJson.IsDouble(jsonVal) THEN							
							lrvoltageP2:= fbJson.GetDouble(jsonVal);									
						END_IF
						jsonVal:= fbJson.FindMember(jsonDoc, 'aenergy');
                        IF fbJson.HasMember(jsonVal, 'total') THEN
                            jsonVal:= fbJson.FindMember(jsonVal, 'total');
                            nValidResCount:= nValidResCount+1;
                            IF fbJson.IsDouble(jsonVal) THEN
                                lraenergyP2:= fbJson.GetDouble(jsonVal);
                            END_IF
						bError:= FALSE;
						END_IF
					END_IF						
				nResCount:= nResCount+1;			
				END_IF
			END_IF
		END_IF
		
		IF NOT fbRequestSwitch2.bError THEN				 
			bGetContentResult:= fbRequestSwitch2.GetContent(pContent:= ADR(sContentS2), nContentSize:= SIZEOF(sContentS2), bSetNullTermination:= TRUE);
			IF fbRequestSwitch2.nStatusCode >= 200 AND fbRequestSwitch2.nStatusCode < 300 THEN
				bGetJsonResult:= FALSE;
				jsonDoc:= fbRequestSwitch2.GetJsonDomContent(fbJson);
				IF jsonDoc <> 0 THEN
					bGetJsonResult:= TRUE;
					IF fbJson.HasMember(jsonDoc, 'output')  THEN
						jsonVal:= fbJson.FindMember(jsonDoc, 'output');
						nValidResCount:= nValidResCount+1;					
						IF fbJson.IsBool(jsonVal) THEN							
							bStateP3:= fbJson.GetBool(jsonVal);									
						END_IF
						jsonVal:= fbJson.FindMember(jsonDoc, 'apower');
						nValidResCount:= nValidResCount+1;
						IF fbJson.IsDouble(jsonVal) THEN							
							lrapowerP3:= fbJson.GetDouble(jsonVal);									
						END_IF
						jsonVal:= fbJson.FindMember(jsonDoc, 'voltage');
						nValidResCount:= nValidResCount+1;					
						IF fbJson.IsDouble(jsonVal) THEN							
							lrvoltageP3:= fbJson.GetDouble(jsonVal);									
						END_IF
						jsonVal:= fbJson.FindMember(jsonDoc, 'aenergy');
                        IF fbJson.HasMember(jsonVal, 'total') THEN
                            jsonVal:= fbJson.FindMember(jsonVal, 'total');
                            nValidResCount:= nValidResCount+1;
                            IF fbJson.IsDouble(jsonVal) THEN
                                lraenergyP3:= fbJson.GetDouble(jsonVal);
                            END_IF
						bError:= FALSE;
						END_IF
					END_IF						
				nResCount:= nResCount+1;			
				END_IF
			END_IF
		END_IF
		
		IF NOT fbRequestSwitch3.bError THEN				 
			bGetContentResult:= fbRequestSwitch3.GetContent(pContent:= ADR(sContentS3), nContentSize:= SIZEOF(sContentS3), bSetNullTermination:= TRUE);
			IF fbRequestSwitch3.nStatusCode >= 200 AND fbRequestSwitch3.nStatusCode < 300 THEN
				bGetJsonResult:= FALSE;
				jsonDoc:= fbRequestSwitch3.GetJsonDomContent(fbJson);
				IF jsonDoc <> 0 THEN
					bGetJsonResult:= TRUE;
					IF fbJson.HasMember(jsonDoc, 'output')  THEN
						jsonVal:= fbJson.FindMember(jsonDoc, 'output');
						nValidResCount:= nValidResCount+1;					
						IF fbJson.IsBool(jsonVal) THEN							
							bStateP4:= fbJson.GetBool(jsonVal);									
						END_IF
						jsonVal:= fbJson.FindMember(jsonDoc, 'apower');
						nValidResCount:= nValidResCount+1;
						IF fbJson.IsDouble(jsonVal) THEN							
							lrapowerP4:= fbJson.GetDouble(jsonVal);									
						END_IF
						jsonVal:= fbJson.FindMember(jsonDoc, 'voltage');
						nValidResCount:= nValidResCount+1;					
						IF fbJson.IsDouble(jsonVal) THEN							
							lrvoltageP4:= fbJson.GetDouble(jsonVal);									
						END_IF
						jsonVal:= fbJson.FindMember(jsonDoc, 'aenergy');
                        IF fbJson.HasMember(jsonVal, 'total') THEN
                            jsonVal:= fbJson.FindMember(jsonVal, 'total');
                            nValidResCount:= nValidResCount+1;
                            IF fbJson.IsDouble(jsonVal) THEN
                                lraenergyP4:= fbJson.GetDouble(jsonVal);
                            END_IF
						bError:= FALSE;
						END_IF
					END_IF						
				nResCount:= nResCount+1;			
				END_IF
			END_IF
		END_IF
		
	nState:= 0;
	bBusy:= FALSE;
		IF bError THEN
			nErrCount:= nErrCount+1;
		END_IF
	END_IF
	
END_CASE

END_FUNCTION_BLOCK

// ---- FBs/FB_Shelly_Pro2PM.TcPOU
FUNCTION_BLOCK FB_Shelly_Pro2PM
VAR_INPUT
	bStart				: BOOL;
	tDelayRequest		: TIME;				//Timer for delay before start with the next read or write Request
	sHostname			: STRING(255);		//Hostname or IP Adress from the Server
	bOnP1				: BOOL;
	bOffP1				: BOOL;
	bOnP2				: BOOL;
	bOffP2				: BOOL;
END_VAR

VAR_OUTPUT
	bValidResult				: BOOL;															//Valid Result received from Server
    bBusy						: BOOL;															//Function is Busy
    bError						: BOOL;															//Error sucess
	bDone						: BOOL;															//True after the decoding from the received Json File
	bConnected					: BOOL;															//Connection to the Server
	hrErrorCode       			: HRESULT;														//Error Result from Http Client
	lrpowerP1					: LREAL;														//Received Value
	lrvoltageP1					: LREAL;														//Received Value
	lrenergyP1					: LREAL;														//Received Value
	lrpowerP2					: LREAL;														//Received Value
	lrvoltageP2					: LREAL;														//Received Value
	lrenergyP2					: LREAL;
	bStateP1					: BOOL;
	bStateP2					: BOOL;
END_VAR

VAR
	fbClient					: FB_IotHttpClient;
	fbHttpGet					: FB_Shelly_Pro2PM_Helper;
	timStartRequest				: TON;															//Timer to Start the Request
	FPStartRequest				: R_TRIG;														//Internal positive Edge
	FPDone						: R_TRIG;														//Internal positive Edge
	FNStart						: F_TRIG;														//Internal negative Edge
	SwitchOnP1					: R_TRIG;
	SwitchOffP1					: R_TRIG;
	SwitchOnP2					: R_TRIG;
	SwitchOffP2					: R_TRIG;
END_VAR

(*------------------------------------------------------------------------------------Configure HTTP Client------------------------------------------------------------------------------------------------------*)

fbClient.sHostName := sHostname;
fbClient.tConnectionTimeout := T#25S;

IF NOT fbClient.bConfigured THEN 
	fbClient.nHostPort:= 80;
	fbClient.bKeepAlive := TRUE;
	fbClient.tConnectionTimeout := T#25S;
END_IF


//Timer to start the Request
FPStartRequest(CLK:= bStart, Q=> );
	timStartRequest(IN:= fbClient.bConfigured AND bStart AND NOT timStartRequest.Q, PT:= tDelayRequest, Q=> , ET=> );
		IF ((timStartRequest.Q AND NOT bBusy) OR (FPStartRequest.Q AND NOT bBusy AND fbClient.bConfigured)) THEN fbHttpGet.bSend := TRUE; END_IF

				
//Http Get Function
fbHttpGet(
	lrapowerP1 => lrpowerP1, 
	lrvoltageP1 => lrvoltageP1, 
	lraenergyP1 => lrenergyP1,
	lrapowerP2 => lrpowerP2, 
	lrvoltageP2 => lrvoltageP2, 
	lraenergyP2 => lrenergyP2,
	bSend:= , 
	fbClient:= fbClient, 
	bBusy=> bBusy, 
	bError=> ,
	sContentS0=> ,
	sContentS1=> ,
	bStateP1=>bStateP1,
	bStateP2=>bStateP2 );


fbHttpGet.bSend := FALSE;

FPDone(CLK:= bDone, Q=> );

fbClient.Execute();

//Error
IF fbHttpGet.bError OR fbClient.bError THEN bError := TRUE; ELSE bError := FALSE; END_IF	
	hrErrorCode := fbClient.hrErrorCode;
	

// Relay Control, Switch P1
SwitchOnP1(CLK:=bOnP1);
IF SwitchOnP1.Q THEN
	fbHttpGet.bSetOnP1 := TRUE;
END_IF

SwitchOffP1(CLK:=bOffP1);
IF SwitchOffP1.Q THEN
	fbHttpGet.bSetOffP1 := TRUE;
END_IF

// Relay Control, Switch P2
SwitchOnP2(CLK:=bOnP2);
IF SwitchOnP2.Q THEN
	fbHttpGet.bSetOnP2 := TRUE;
END_IF

SwitchOffP2(CLK:=bOffP2);
IF SwitchOffP2.Q THEN
	fbHttpGet.bSetOffP2 := TRUE;
END_IF

END_FUNCTION_BLOCK

// ---- FBs/FB_Shelly_Pro2PM_Helper.TcPOU
FUNCTION_BLOCK FB_Shelly_Pro2PM_Helper
VAR_INPUT
	bSend			: BOOL;
	bSetOnP1		: BOOL;
	bSetOffP1		: BOOL;
	bSetOnP2		: BOOL;
	bSetOffP2		: BOOL;
END_VAR

VAR_IN_OUT
	fbClient		: FB_IotHttpClient;
END_VAR

VAR_OUTPUT
	bBusy			: BOOL;
	bError			: BOOL;
	bStateP1		: BOOL;
	bStateP2		: BOOL;
	lrapowerP1		: LREAL;
	lrvoltageP1		: LREAL;
	lraenergyP1		: LREAL;
	lrapowerP2		: LREAL;
	lrvoltageP2		: LREAL;
	lraenergyP2		: LREAL;
END_VAR

VAR
	fbRequestSwitch0	: FB_IotHttpRequest;
	fbRequestSwitch1	: FB_IotHttpRequest;
	RisingEdge			: R_TRIG;
	RisingEdgeSetOnP1	: R_TRIG;
	RisingEdgeSetOffP1	: R_TRIG;
	RisingEdgeSetOnP2	: R_TRIG;
	RisingEdgeSetOffP2	: R_TRIG;
	fbJson				: FB_JsonDomParser;
	nState				: UDINT;
	timTimeout			: TON;
	tTimeOut			: TIME := T#30S;
	timTimeoutSwitch	: TON;
	tTimeOutSwitch		: TIME := T#5S;
	bGetContentResult	: BOOL;
	sContentS0			: STRING(511);
	sContentS1			: STRING(511);
	
	bGetJsonResult		: BOOL;
	jsonDoc				: SJsonValue;
	jsonVal				: SJsonValue;
	
	nReqCount			: UDINT;	
	nResCount			: UDINT;
	nValidResCount		: UDINT;
	nErrCount			: UDINT;
END_VAR

//Timer for Timeout
timTimeout(IN:= nState = 1 AND bBusy, PT:= tTimeOut, Q=> , ET=> );
	IF timTimeout.Q THEN 
		nState := 0;
		bBusy := FALSE;
	END_IF
	
timTimeoutSwitch(IN:= bSetOnP1 OR bSetOffP1 OR bSetOnP2 OR bSetOffP2, PT:= tTimeOut, Q=> , ET=> );
	IF timTimeoutSwitch.Q THEN 
		bSetOnP1 := FALSE;
		bSetOffP1 := FALSE;
		bSetOnP2 := FALSE;
		bSetOffP2 := FALSE;
	END_IF

RisingEdge(CLK:= bSend );
RisingEdgeSetOnP1(CLK:= bSetOnP1 );
RisingEdgeSetOffP1(CLK:= bSetOffP1 );
RisingEdgeSetOnP2(CLK:= bSetOnP2 );
RisingEdgeSetOffP2(CLK:= bSetOffP2 );

CASE nState OF
0:	
	IF RisingEdge.Q THEN 
		IF
			fbRequestSwitch0.SendRequest(sUri:='/rpc/Switch.GetStatus?id=0', fbClient:=fbClient, eRequestType:=ETcIotHttpRequestType.HTTP_Get, 0, 0, 0) AND
			fbRequestSwitch1.SendRequest(sUri:='/rpc/Switch.GetStatus?id=1', fbClient:=fbClient, eRequestType:=ETcIotHttpRequestType.HTTP_Get, 0, 0, 0) THEN
			nState:= 1;
			nReqCount:= nReqCount+1;
			bBusy:= TRUE;
			bError:= FALSE;
		END_IF					
	END_IF
	
	IF RisingEdgeSetOnP1.Q THEN 
		IF
			fbRequestSwitch0.SendRequest(sUri:='/rpc/Switch.Set?id=0&on=true', fbClient:=fbClient, eRequestType:=ETcIotHttpRequestType.HTTP_Get, 0, 0, 0) THEN				
			bSetOnP1 := FALSE;
			nState:= 1;
			bBusy:= TRUE;
			bError:= FALSE;
		END_IF					
	END_IF
	
	IF RisingEdgeSetOffP1.Q THEN 
		IF
			fbRequestSwitch0.SendRequest(sUri:='/rpc/Switch.Set?id=0&on=false', fbClient:=fbClient, eRequestType:=ETcIotHttpRequestType.HTTP_Get, 0, 0, 0) THEN				
			bSetOffP1 := FALSE;
			nState:= 1;
			bBusy:= TRUE;
			bError:= FALSE;
		END_IF					
	END_IF
	
	IF RisingEdgeSetOnP2.Q THEN 
		IF
			fbRequestSwitch1.SendRequest(sUri:='/rpc/Switch.Set?id=1&on=true', fbClient:=fbClient, eRequestType:=ETcIotHttpRequestType.HTTP_Get, 0, 0, 0) THEN				
			bSetOnP2 := FALSE;
			nState:= 1;
			bBusy:= TRUE;
			bError:= FALSE;
		END_IF					
	END_IF
	
	IF RisingEdgeSetOffP2.Q THEN 
		IF
			fbRequestSwitch1.SendRequest(sUri:='/rpc/Switch.Set?id=1&on=false', fbClient:=fbClient, eRequestType:=ETcIotHttpRequestType.HTTP_Get, 0, 0, 0) THEN				
			bSetOffP2 := FALSE;
			nState:= 1;
			bBusy:= TRUE;
			bError:= FALSE;
		END_IF					
	END_IF
	
1:
	IF NOT fbRequestSwitch0.bBusy AND NOT fbRequestSwitch1.bBusy THEN
		bError:= TRUE;
		
		IF NOT fbRequestSwitch0.bError THEN				 
			bGetContentResult:= fbRequestSwitch0.GetContent(pContent:= ADR(sContentS0), nContentSize:= SIZEOF(sContentS0), bSetNullTermination:= TRUE);
			IF fbRequestSwitch0.nStatusCode >= 200 AND fbRequestSwitch0.nStatusCode < 300 THEN
				bGetJsonResult:= FALSE;
				jsonDoc:= fbRequestSwitch0.GetJsonDomContent(fbJson);
				IF jsonDoc <> 0 THEN
					bGetJsonResult:= TRUE;
					IF fbJson.HasMember(jsonDoc, 'output')  THEN
						jsonVal:= fbJson.FindMember(jsonDoc, 'output');
						nValidResCount:= nValidResCount+1;					
						IF fbJson.IsBool(jsonVal) THEN							
							bStateP1:= fbJson.GetBool(jsonVal);									
						END_IF
						jsonVal:= fbJson.FindMember(jsonDoc, 'apower');
						nValidResCount:= nValidResCount+1;
						IF fbJson.IsDouble(jsonVal) THEN							
							lrapowerP1:= fbJson.GetDouble(jsonVal);									
						END_IF
						jsonVal:= fbJson.FindMember(jsonDoc, 'voltage');
						nValidResCount:= nValidResCount+1;					
						IF fbJson.IsDouble(jsonVal) THEN							
							lrvoltageP1:= fbJson.GetDouble(jsonVal);									
						END_IF
						jsonVal:= fbJson.FindMember(jsonDoc, 'aenergy');
                        IF fbJson.HasMember(jsonVal, 'total') THEN
                            jsonVal:= fbJson.FindMember(jsonVal, 'total');
                            nValidResCount:= nValidResCount+1;
                            IF fbJson.IsDouble(jsonVal) THEN
                                lraenergyP1:= fbJson.GetDouble(jsonVal);
                            END_IF
						bError:= FALSE;
						END_IF
					END_IF						
				nResCount:= nResCount+1;			
				END_IF
			END_IF
		END_IF
		
		IF NOT fbRequestSwitch1.bError THEN				 
			bGetContentResult:= fbRequestSwitch1.GetContent(pContent:= ADR(sContentS1), nContentSize:= SIZEOF(sContentS1), bSetNullTermination:= TRUE);
			IF fbRequestSwitch1.nStatusCode >= 200 AND fbRequestSwitch1.nStatusCode < 300 THEN
				bGetJsonResult:= FALSE;
				jsonDoc:= fbRequestSwitch1.GetJsonDomContent(fbJson);
				IF jsonDoc <> 0 THEN
					bGetJsonResult:= TRUE;
					IF fbJson.HasMember(jsonDoc, 'output')  THEN
						jsonVal:= fbJson.FindMember(jsonDoc, 'output');
						nValidResCount:= nValidResCount+1;					
						IF fbJson.IsBool(jsonVal) THEN							
							bStateP2:= fbJson.GetBool(jsonVal);									
						END_IF
						jsonVal:= fbJson.FindMember(jsonDoc, 'apower');
						nValidResCount:= nValidResCount+1;
						IF fbJson.IsDouble(jsonVal) THEN							
							lrapowerP2:= fbJson.GetDouble(jsonVal);									
						END_IF
						jsonVal:= fbJson.FindMember(jsonDoc, 'voltage');
						nValidResCount:= nValidResCount+1;					
						IF fbJson.IsDouble(jsonVal) THEN							
							lrvoltageP2:= fbJson.GetDouble(jsonVal);									
						END_IF
						jsonVal:= fbJson.FindMember(jsonDoc, 'aenergy');
                        IF fbJson.HasMember(jsonVal, 'total') THEN
                            jsonVal:= fbJson.FindMember(jsonVal, 'total');
                            nValidResCount:= nValidResCount+1;
                            IF fbJson.IsDouble(jsonVal) THEN
                                lraenergyP2:= fbJson.GetDouble(jsonVal);
                            END_IF
						bError:= FALSE;
						END_IF
					END_IF						
				nResCount:= nResCount+1;			
				END_IF
			END_IF
		END_IF
		
	nState:= 0;
	bBusy:= FALSE;
		IF bError THEN
			nErrCount:= nErrCount+1;
		END_IF
	END_IF
	
END_CASE

END_FUNCTION_BLOCK

// ---- POUs/prgComEffIO.TcPOU
PROGRAM prgComEffIO
VAR
	fbCom		: FB_MqttCommunicator_V2;
	f_Trig_HB: f_trig;
	stringArray_Last_HB: ARRAY[0..50] OF STRING(30);
	intCount: INT;
	time_Temp: TIME;
	time_HB: TIME:= T#15S;
END_VAR

fbCom(
	bConnect:= TRUE, 
	sUserName:= 'b472a324-06e3-4d07-96cf-574b1847d8ff', 
	sUserPassword:= '5b687dd8-7c3c-4e3c-8272-e8ed6dc08177', 
	strAuthKey:= 'EIO08031879806', 
	eSavePositionCertificate:= eSavePositionOnPLC.ePostionHardDisk, 
	time_HeartBeat_sec := time_HB,
	bConnected=> , 
	bError=> , 
	hrErrorCode=> , 
	eConnectionState=> , 
	eErrorMessage_Out=> );
	
f_Trig_HB(CLK :=  fbCom.bHBSending);



prg_SystemTime();

IF f_Trig_HB.Q THEN
	stringArray_Last_HB[intCount] := prg_SystemTime.stringSystemTime_ms;
	intCount := intCount+1;
	IF intCount>50 OR intCount<0 THEN
		intCount:=0;
	END_IF
	stringArray_Last_HB[intCount] := '';
END_IF

time_Temp := fbCom.fbTimerHB.ET;

END_PROGRAM
